	IF i16_anfangspos_mit_tzk[no] < 0 OR i16_endpos_mit_tzk[no] < 0 OR i16_anfangspos_mit_tzk[no] >= 360 OR i16_endpos_mit_tzk[no] >= 360 THEN
		 (* Fehlerfälle  mit Abbruch*)
		sm_positionseingabe := TRUE;
		EXIT; (* Schleifenabbruch *)
	ELSE (* Winkel sind o.k. und der Nocken wird bearbeitet -> ON/OFF *)
		sm_positionseingabe := FALSE;
		IF i16_anfangspos_mit_tzk[no] <> i16_endpos_mit_tzk[no] THEN
			(* Nocken setzen *)
			(* Anfangswinkel ist kleiner Endwinkel *)
			b_setzustand_anfang_kleiner_ende[no] := i16_anfangspos_mit_tzk[no] < i16_endpos_mit_tzk[no] AND
												i16_aktuelle_pos >= i16_anfangspos_mit_tzk[no] AND
												i16_aktuelle_pos <= i16_endpos_mit_tzk[no];
			(* Anfangswinkel ist grösser Endwinkel *)
			b_setzustand_anfang_groesser_ende[no] := i16_anfangspos_mit_tzk[no] > i16_endpos_mit_tzk[no] AND
												(i16_aktuelle_pos >= i16_anfangspos_mit_tzk[no] OR
												i16_aktuelle_pos <= i16_endpos_mit_tzk[no]);

			(* Nocken ist gültig, d.h. wurde von der Maschine oder Bediener aktiviert *)
			IF	arr_nocken[no].b_camvalid AND
				(b_setzustand_anfang_kleiner_ende[no] OR b_setzustand_anfang_groesser_ende[no]) AND
				((b_verfahrrichtung_positiv AND arr_nocken[no].b_eff_direction_pos) OR	(* positive Drehrichtung und positive Wirkrichtung ist freigegeben *)
				(b_verfahrrichtung_negativ AND arr_nocken[no].b_eff_direction_neg)) 		(* negative Drehrichtung und negative Wirkrichtung ist freigegeben *)
				THEN
					arr_nocken[no].b_nockenzustand := TRUE;
			END_IF

			(* Nocken zurücksetzen *)
			(* Anfangswinkel ist kleiner Endwinkel *)
			b_resetzustand_anfang_kleiner_ende[no] := i16_anfangspos_mit_tzk[no] < i16_endpos_mit_tzk[no] AND
													(i16_aktuelle_pos < i16_anfangspos_mit_tzk[no] OR
													i16_aktuelle_pos  > i16_endpos_mit_tzk[no]);
			(* Anfangswinkel ist grösser Endwinkel *)
			b_resetzustand_anfang_groesser_ende[no] := i16_anfangspos_mit_tzk[no] > i16_endpos_mit_tzk[no] AND
													i16_aktuelle_pos < i16_anfangspos_mit_tzk[no] AND
													i16_aktuelle_pos > i16_endpos_mit_tzk[no];

			(* Nocken ist ungültig, d.h. wurde von der Maschine oder Bediener deaktiviert *)
			IF	NOT arr_nocken[no].b_camvalid OR
				(b_resetzustand_anfang_kleiner_ende[no] OR b_resetzustand_anfang_groesser_ende[no])
				THEN
					arr_nocken[no].b_nockenzustand := FALSE;
			END_IF
		ELSE
			(* Anfang = Ende -> Nocken ist false *)
			arr_nocken[no].b_nockenzustand := FALSE;
		END_IF
	END_IF

	(* Aktive Nocken auf ihre Spuren setzen *)
	IF arr_nocken[no].b_camvalid AND arr_nocken[no].b_nockenzustand THEN
		arr_spur[arr_nocken[no].i16_track_no] := TRUE;
	END_IF
END_FOR

IF st_config.b_config_fertig THEN
	(* Fehlermeldungen und Betriebsmeldungen ab dem Startindex in die globalen Meldungsarrays schreiben *)
	garr_stoermeldungen[st_config.i16_meld_startindex + 0] := sm_positionseingabe;
	garr_stoermeldungen[st_config.i16_meld_startindex + 1] := sm_vorsteuerung;
	garr_stoermeldungen[st_config.i16_meld_startindex + 2] := FALSE;
	garr_stoermeldungen[st_config.i16_meld_startindex + 3] := FALSE;
	garr_stoermeldungen[st_config.i16_meld_startindex + 4] := FALSE;
	garr_stoermeldungen[st_config.i16_meld_startindex + 5] := FALSE;
	garr_stoermeldungen[st_config.i16_meld_startindex + 6] := FALSE;
	garr_stoermeldungen[st_config.i16_meld_startindex + 7] := FALSE;
	garr_stoermeldungen[st_config.i16_meld_startindex + 8] := FALSE;
	garr_stoermeldungen[st_config.i16_meld_startindex + 9] := FALSE;
	garr_stoermeldungen[st_config.i16_meld_startindex + 10] := FALSE;
	garr_stoermeldungen[st_config.i16_meld_startindex + 11] := FALSE;
	garr_stoermeldungen[st_config.i16_meld_startindex + 12] := FALSE;
	garr_stoermeldungen[st_config.i16_meld_startindex + 13] := FALSE;
	garr_stoermeldungen[st_config.i16_meld_startindex + 14] := FALSE;
	garr_stoermeldungen[st_config.i16_meld_startindex + 15] := FALSE;
	garr_stoermeldungen[st_config.i16_meld_startindex + 16] := FALSE;
	garr_stoermeldungen[st_config.i16_meld_startindex + 17] := FALSE;
	garr_stoermeldungen[st_config.i16_meld_startindex + 18] := FALSE;
	garr_stoermeldungen[st_config.i16_meld_startindex + 19] := FALSE;
	
	garr_betriebsmeldungen[st_config.i16_meld_startindex + 0] := FALSE;
	garr_betriebsmeldungen[st_config.i16_meld_startindex + 1] := FALSE;
	garr_betriebsmeldungen[st_config.i16_meld_startindex + 2] := FALSE;
	garr_betriebsmeldungen[st_config.i16_meld_startindex + 3] := FALSE;
	garr_betriebsmeldungen[st_config.i16_meld_startindex + 4] := FALSE;
	garr_betriebsmeldungen[st_config.i16_meld_startindex + 5] := FALSE;
	garr_betriebsmeldungen[st_config.i16_meld_startindex + 6] := FALSE;
	garr_betriebsmeldungen[st_config.i16_meld_startindex + 7] := FALSE;
	garr_betriebsmeldungen[st_config.i16_meld_startindex + 8] := FALSE;
	garr_betriebsmeldungen[st_config.i16_meld_startindex + 9] := FALSE;
	garr_betriebsmeldungen[st_config.i16_meld_startindex + 10] := FALSE;
	garr_betriebsmeldungen[st_config.i16_meld_startindex + 11] := FALSE;
	garr_betriebsmeldungen[st_config.i16_meld_startindex + 12] := FALSE;
	garr_betriebsmeldungen[st_config.i16_meld_startindex + 13] := FALSE;
	garr_betriebsmeldungen[st_config.i16_meld_startindex + 14] := FALSE;
	garr_betriebsmeldungen[st_config.i16_meld_startindex + 15] := FALSE;
	garr_betriebsmeldungen[st_config.i16_meld_startindex + 16] := FALSE;
	garr_betriebsmeldungen[st_config.i16_meld_startindex + 17] := FALSE;
	garr_betriebsmeldungen[st_config.i16_meld_startindex + 18] := FALSE;
	garr_betriebsmeldungen[st_config.i16_meld_startindex + 19] := FALSE;
END_IF
END_FUNCTION_BLOCK

(* POU EPT Lib/Funktionsbausteine/Nockenschaltwerke/NSW_LREAL/ST_Nockenschaltwerk_lreal, ST *)
FUNCTION_BLOCK ST_Nockenschaltwerk_lreal
VAR_INPUT
	r_achsposition							: LREAL;
	r_achsgeschwindigkeit						: LREAL;
	i16_verfahrrichtung_achse_extern			: INT;
	b_verfahrrichtungsauswertung_extern			: BOOL;
	i16_art_der_achse							: enum_ecd_typ;
	st_config									: struct_config;
END_VAR
VAR_IN_OUT
	st_visu									: struct_visu;
	arr_nocken								: ARRAY [0..MAX_NOCKENGERUEST] OF struct_nocken_lreal;
END_VAR
VAR_OUTPUT
END_VAR
VAR
	b_first_cycle 								: BOOL := TRUE;
	r_aktuelle_pos 							: T_FIX16;
	r_alte_pos	 							: T_FIX16;
	b_verfahrrichtung_positiv 					: BOOL := FALSE;
	b_verfahrrichtung_negativ					: BOOL := FALSE;
	r_zeit_fuer_1einheit						: LREAL := 0.0;
	r_anfangspos_mit_tzk 						: ARRAY [0..MAX_NOCKENGERUEST] OF LREAL := 0.0;
	r_endpos_mit_tzk 							: ARRAY [0..MAX_NOCKENGERUEST] OF LREAL := 0.0;
	r_vorsteuerpos_max						: LREAL := 0.0;
	i16_verfahrrichtung_achse_intern				: INT := 0;
	sm_positionseingabe						: BOOL := FALSE;
	sm_vorsteuerung							: BOOL := FALSE;
	sp, no									: UINT := 0;
	arr_spur									: ARRAY [0..MAX_NOCKENGERUEST] OF BOOL;
	b_setzustand_anfang_kleiner_ende			: ARRAY [0..MAX_NOCKENGERUEST] OF BOOL;
	b_setzustand_anfang_groesser_ende		: ARRAY [0..MAX_NOCKENGERUEST] OF BOOL;
	b_resetzustand_anfang_kleiner_ende		: ARRAY [0..MAX_NOCKENGERUEST] OF BOOL;
	b_resetzustand_anfang_groesser_ende		: ARRAY [0..MAX_NOCKENGERUEST] OF BOOL;
END_VAR
(* Funktionsbaustein Nockenschaltwerk *)
(* Funktion für lineare und rotatorische Achsen *)
CASE i16_art_der_achse  OF
1:	(* Linearachse *)
	IF b_first_cycle THEN
		b_first_cycle := FALSE;

		(* Setze Drehrichtung Positiv. Da wenn beide Drehrichtungen nicht gesetzt sind, keine Nocke aktiv wird *)
		r_vorsteuerpos_max := 100.0;
		b_verfahrrichtung_positiv := TRUE;
		b_verfahrrichtung_negativ := FALSE;
		r_alte_pos := r_aktuelle_pos;
	END_IF

	(* Aktuelle Position für weitere Komponenten zur Verfügung stellen *)
	r_aktuelle_pos := LREAL_TO_FIX16(r_achsposition,2);

	(* Verfahrrichtung überwachen *)
	IF FIX16_TO_LREAL(r_aktuelle_pos) > FIX16_TO_LREAL(r_alte_pos) THEN
		i16_verfahrrichtung_achse_intern := 1;
		r_alte_pos := r_aktuelle_pos;
	ELSIF FIX16_TO_LREAL(r_aktuelle_pos) < FIX16_TO_LREAL(r_alte_pos) THEN
		i16_verfahrrichtung_achse_intern := -1;
		r_alte_pos := r_aktuelle_pos;
	END_IF

	IF b_verfahrrichtungsauswertung_extern THEN
		IF i16_verfahrrichtung_achse_extern = 1 THEN
			b_verfahrrichtung_positiv := TRUE;
			b_verfahrrichtung_negativ := FALSE;
		ELSIF i16_verfahrrichtung_achse_extern = -1 THEN
			b_verfahrrichtung_positiv := FALSE;
			b_verfahrrichtung_negativ := TRUE;
		END_IF
	ELSE
		IF i16_verfahrrichtung_achse_intern = 1 THEN
			b_verfahrrichtung_positiv := TRUE;
			b_verfahrrichtung_negativ := FALSE;
		ELSIF i16_verfahrrichtung_achse_intern = -1 THEN
			b_verfahrrichtung_positiv := FALSE;
			b_verfahrrichtung_negativ := TRUE;
		END_IF
	END_IF

	IF r_achsgeschwindigkeit >= 1.0 THEN
		r_zeit_fuer_1einheit := 0.001 * r_achsgeschwindigkeit;		(* REAL-Zahl in ms *)
	ELSE
		r_zeit_fuer_1einheit := 0.0;
	END_IF

	(* Totzeitkompensation durch Vorsteuerung *)
	FOR no := 0  TO SIZEOF (arr_nocken)/SIZEOF(arr_nocken[0]) -1 DO
		(* Berechnung der Vorsteuerposition *)
		 arr_nocken[no].r_vorsteuerpos :=  (TIME_TO_LREAL(arr_nocken[no].t_vorsteuerzeit)) * r_zeit_fuer_1einheit;
		IF  arr_nocken[no].r_vorsteuerpos >= r_vorsteuerpos_max THEN
			 arr_nocken[no].r_vorsteuerpos := 0.0;
			sm_vorsteuerung := TRUE;
		ELSE
			sm_vorsteuerung := FALSE;
		END_IF

		(* Nockentoleranz mit Berücksichtigung der Vorsteuerzeit für Anfangswinkel*)
		r_anfangspos_mit_tzk[no] := arr_nocken[no].r_cam_begin - arr_nocken[no].r_vorsteuerpos;
		(* Nockentoleranz mit Berücksichtigung der Vorsteuerzeit für Endwinkel*)
		r_endpos_mit_tzk[no] := arr_nocken[no].r_cam_end - arr_nocken[no].r_vorsteuerpos;

		IF r_anfangspos_mit_tzk[no] <> r_endpos_mit_tzk[no] THEN
			(* Nocken setzen *)
			(* Anfangsposition ist kleiner Endposition *)
			b_setzustand_anfang_kleiner_ende[no] := r_anfangspos_mit_tzk[no] < r_endpos_mit_tzk[no] AND
													FIX16_TO_LREAL(r_aktuelle_pos) >= r_anfangspos_mit_tzk[no] AND
													FIX16_TO_LREAL(r_aktuelle_pos) <= r_endpos_mit_tzk[no];
			(* Anfangsposition ist grösser Endposition *)
			b_setzustand_anfang_groesser_ende[no] := r_anfangspos_mit_tzk[no] > r_endpos_mit_tzk[no] AND
													FIX16_TO_LREAL(r_aktuelle_pos) <= r_anfangspos_mit_tzk[no] AND
													FIX16_TO_LREAL(r_aktuelle_pos) >= r_endpos_mit_tzk[no];
	
			(* Nocken ist gültig, d.h. wurde von der Maschine oder Bediener aktiviert *)
			IF	arr_nocken[no].b_camvalid AND
				(b_setzustand_anfang_kleiner_ende[no] OR b_setzustand_anfang_groesser_ende[no]) AND
				((b_verfahrrichtung_positiv AND arr_nocken[no].b_eff_direction_pos) OR	(* positive Drehrichtung und positive Wirkrichtung ist freigegeben *)
				(b_verfahrrichtung_negativ AND arr_nocken[no].b_eff_direction_neg)) 		(* negative Drehrichtung und negative Wirkrichtung ist freigegeben *)
				THEN
					arr_nocken[no].b_nockenzustand := TRUE;
			END_IF
	
			(* Nocken zurücksetzen *)
			(* Anfangswinkel ist kleiner Endwinkel *)
			b_resetzustand_anfang_kleiner_ende[no] := r_anfangspos_mit_tzk[no] < r_endpos_mit_tzk[no] AND
													(FIX16_TO_LREAL(r_aktuelle_pos) < r_anfangspos_mit_tzk[no] OR
													FIX16_TO_LREAL(r_aktuelle_pos)  > r_endpos_mit_tzk[no]);
			(* Anfangswinkel ist grösser Endwinkel *)
			b_resetzustand_anfang_groesser_ende[no] := r_anfangspos_mit_tzk[no] > r_endpos_mit_tzk[no] AND
													(FIX16_TO_LREAL(r_aktuelle_pos) > r_anfangspos_mit_tzk[no] OR
													FIX16_TO_LREAL(r_aktuelle_pos) < r_endpos_mit_tzk[no]);
	
			(* Nocken ist ungültig, d.h. wurde von der Maschine oder Bediener deaktiviert *)
			IF	NOT arr_nocken[no].b_camvalid OR
				b_resetzustand_anfang_kleiner_ende[no] OR
				b_resetzustand_anfang_groesser_ende[no] OR
				(* Zusatzbedingung für Nockenzustand rücksetzen ist nur bei Linearachsen sinnvoll *)
				(b_verfahrrichtung_positiv AND NOT arr_nocken[no].b_eff_direction_pos AND arr_nocken[no].b_eff_direction_neg) OR	(* positive Drehrichtung und positive Wirkrichtung ist freigegeben *)
				(b_verfahrrichtung_negativ AND NOT arr_nocken[no].b_eff_direction_neg AND arr_nocken[no].b_eff_direction_pos)		(* negative Drehrichtung und negative Wirkrichtung ist freigegeben *)
				THEN
					arr_nocken[no].b_nockenzustand := FALSE;
			END_IF
		ELSE
			(* Anfang = Ende -> Nocken ist false *)
			arr_nocken[no].b_nockenzustand := FALSE;
		END_IF
	END_FOR

	(* Erst alle Spuren reset *)
	FOR sp := 0  TO SIZEOF (arr_spur)-1 DO
		arr_spur[sp] :=FALSE;
	END_FOR
	
	(* Dann aktive Nocken auf ihre Spuren setzen *)
	FOR no := 0  TO SIZEOF (arr_nocken)/SIZEOF(arr_nocken[0])-1 DO
		IF arr_nocken[no].b_camvalid AND arr_nocken[no].b_nockenzustand THEN
			arr_spur[arr_nocken[no].i16_track_no] := TRUE;
		END_IF
	END_FOR

2:	(* Rotatorische Achse *)
	IF b_first_cycle THEN
		b_first_cycle := FALSE;

		(* Setze Drehrichtung Positiv. Da wenn beide Drehrichtungen nicht gesetzt sind, keine Nocke aktiv wird *)
		r_vorsteuerpos_max := 60.0;
		b_verfahrrichtung_positiv := TRUE;
		b_verfahrrichtung_negativ := FALSE;
		r_alte_pos := r_aktuelle_pos;
	END_IF

	(* Aktuelle Position für weitere Komponenten zur Verfügung stellen *)
	r_aktuelle_pos := LREAL_TO_FIX16(r_achsposition,2);

	(* Verfahrrichtung überwachen *)
	IF FIX16_TO_LREAL(r_aktuelle_pos) > FIX16_TO_LREAL(r_alte_pos) THEN
		i16_verfahrrichtung_achse_intern := 1;
		r_alte_pos := r_aktuelle_pos;
	ELSIF FIX16_TO_LREAL(r_aktuelle_pos) < FIX16_TO_LREAL(r_alte_pos) THEN
		i16_verfahrrichtung_achse_intern := -1;
		r_alte_pos := r_aktuelle_pos;
	END_IF

	IF b_verfahrrichtungsauswertung_extern THEN
		IF i16_verfahrrichtung_achse_extern = 1 THEN
			b_verfahrrichtung_positiv := TRUE;
			b_verfahrrichtung_negativ := FALSE;
		ELSIF i16_verfahrrichtung_achse_extern = -1 THEN
			b_verfahrrichtung_positiv := FALSE;
			b_verfahrrichtung_negativ := TRUE;
		END_IF
	ELSE
		IF i16_verfahrrichtung_achse_intern = 1 THEN
			b_verfahrrichtung_positiv := TRUE;
			b_verfahrrichtung_negativ := FALSE;
		ELSIF i16_verfahrrichtung_achse_intern = -1 THEN
			b_verfahrrichtung_positiv := FALSE;
			b_verfahrrichtung_negativ := TRUE;
		END_IF
	END_IF

	IF r_achsgeschwindigkeit >= 1.0 THEN
		(* 0.006 = 360Grad / (60sec * 1000ms) *)
		r_zeit_fuer_1einheit := 0.006 * r_achsgeschwindigkeit;	(* REAL-Zahl in ms *)
	ELSE
		r_zeit_fuer_1einheit := 0.0;
	END_IF

	(* Totzeitkompensation durch Vorsteuerung *)
	FOR no := 0  TO SIZEOF (arr_nocken)/SIZEOF(arr_nocken[0]) -1 DO
		(* Berechnung des Vorsteuerwinkels *)
		arr_nocken[no].r_vorsteuerpos :=  (TIME_TO_LREAL(arr_nocken[no].t_vorsteuerzeit)) * r_zeit_fuer_1einheit;
		IF  arr_nocken[no].r_vorsteuerpos >= r_vorsteuerpos_max THEN
			 arr_nocken[no].r_vorsteuerpos := 0.0;
			sm_vorsteuerung := TRUE;
		ELSE
			sm_vorsteuerung := FALSE;
		END_IF

		(* Nockentoleranz mit Berücksichtigung der Vorsteuerzeit für Anfangswinkel*)
		r_anfangspos_mit_tzk[no] := arr_nocken[no].r_cam_begin -  arr_nocken[no].r_vorsteuerpos;
		IF r_anfangspos_mit_tzk[no] > 360.0 THEN
			r_anfangspos_mit_tzk[no] := r_anfangspos_mit_tzk[no] - 360.0;
		ELSIF r_anfangspos_mit_tzk[no] < 0.0 THEN
			r_anfangspos_mit_tzk[no] := r_anfangspos_mit_tzk[no] + 360.0;
		END_IF
		(* Nockentoleranz mit Berücksichtigung der Vorsteuerzeit für Endwinkel*)
		r_endpos_mit_tzk[no] := arr_nocken[no].r_cam_end -  arr_nocken[no].r_vorsteuerpos;
		IF r_endpos_mit_tzk[no] > 360.0 THEN
			r_endpos_mit_tzk[no] := r_endpos_mit_tzk[no] - 360.0;
		ELSIF r_endpos_mit_tzk[no] < 0.0 THEN
			r_endpos_mit_tzk[no] := r_endpos_mit_tzk[no] + 360.0;
		END_IF
	
		IF r_anfangspos_mit_tzk[no] < 0.0 OR r_endpos_mit_tzk[no] < 0.0 OR r_anfangspos_mit_tzk[no] >= 360.0 OR r_endpos_mit_tzk[no] >= 360.0 THEN
			 (* Fehlerfälle  mit Abbruch*)
			sm_positionseingabe := TRUE;
			EXIT; (* Schleifenabbruch *)
		ELSE (* Winkel sind o.k. und der Nocken wird bearbeitet -> ON/OFF *)
			sm_positionseingabe := FALSE;
			IF r_anfangspos_mit_tzk[no] <> r_endpos_mit_tzk[no] THEN
				(* Nocken setzen *)
				(* Anfangswinkel ist kleiner Endwinkel *)
				b_setzustand_anfang_kleiner_ende[no] := r_anfangspos_mit_tzk[no] < r_endpos_mit_tzk[no] AND
													FIX16_TO_LREAL(r_aktuelle_pos) >= r_anfangspos_mit_tzk[no] AND
													FIX16_TO_LREAL(r_aktuelle_pos) <= r_endpos_mit_tzk[no];
				(* Anfangswinkel ist grösser Endwinkel *)
				b_setzustand_anfang_groesser_ende[no] := r_anfangspos_mit_tzk[no] > r_endpos_mit_tzk[no] AND
													(FIX16_TO_LREAL(r_aktuelle_pos) >= r_anfangspos_mit_tzk[no] OR
													FIX16_TO_LREAL(r_aktuelle_pos) <= r_endpos_mit_tzk[no]);

				(* Nocken ist gültig, d.h. wurde von der Maschine oder Bediener aktiviert *)
				IF	arr_nocken[no].b_camvalid AND
					(b_setzustand_anfang_kleiner_ende[no] OR b_setzustand_anfang_groesser_ende[no]) AND
					((b_verfahrrichtung_positiv AND arr_nocken[no].b_eff_direction_pos) OR	(* positive Drehrichtung und positive Wirkrichtung ist freigegeben *)
					(b_verfahrrichtung_negativ AND arr_nocken[no].b_eff_direction_neg)) 		(* negative Drehrichtung und negative Wirkrichtung ist freigegeben *)
					THEN
						arr_nocken[no].b_nockenzustand := TRUE;
				END_IF

				(* Nocken zurücksetzen *)
				(* Anfangswinkel ist kleiner Endwinkel *)
				b_resetzustand_anfang_kleiner_ende[no] := r_anfangspos_mit_tzk[no] < r_endpos_mit_tzk[no] AND
														(FIX16_TO_LREAL(r_aktuelle_pos) < r_anfangspos_mit_tzk[no] OR
														FIX16_TO_LREAL(r_aktuelle_pos)  > r_endpos_mit_tzk[no]);
				(* Anfangswinkel ist grösser Endwinkel *)
				b_resetzustand_anfang_groesser_ende[no] := r_anfangspos_mit_tzk[no] > r_endpos_mit_tzk[no] AND
														FIX16_TO_LREAL(r_aktuelle_pos) < r_anfangspos_mit_tzk[no] AND
														FIX16_TO_LREAL(r_aktuelle_pos) > r_endpos_mit_tzk[no];

				(* Nocken ist ungültig, d.h. wurde von der Maschine oder Bediener deaktiviert *)
				IF	NOT arr_nocken[no].b_camvalid OR
					(b_resetzustand_anfang_kleiner_ende[no] OR b_resetzustand_anfang_groesser_ende[no])
					THEN
						arr_nocken[no].b_nockenzustand := FALSE;
				END_IF
			ELSE
				(* Anfang = Ende -> Nocken ist false *)
				arr_nocken[no].b_nockenzustand := FALSE;
			END_IF
		END_IF
	END_FOR

	(* Erst alle Spuren reset *)
	FOR sp := 0  TO SIZEOF (arr_spur)-1 DO
		arr_spur[sp] :=FALSE;
	END_FOR

	(* Dann aktive Nocken auf ihre Spuren setzen *)
	FOR no := 0  TO SIZEOF (arr_nocken)/SIZEOF(arr_nocken[0])-1 DO
		IF arr_nocken[no].b_camvalid AND arr_nocken[no].b_nockenzustand THEN
			arr_spur[arr_nocken[no].i16_track_no] := TRUE;
		END_IF
	END_FOR
END_CASE

IF st_config.b_config_fertig THEN
	(* Fehlermeldungen und Betriebsmeldungen ab dem Startindex in die globalen Meldungsarrays schreiben *)
	garr_stoermeldungen[st_config.i16_meld_startindex + 0] := sm_positionseingabe;
	garr_stoermeldungen[st_config.i16_meld_startindex + 1] := sm_vorsteuerung;
	garr_stoermeldungen[st_config.i16_meld_startindex + 2] := FALSE;
	garr_stoermeldungen[st_config.i16_meld_startindex + 3] := FALSE;
	garr_stoermeldungen[st_config.i16_meld_startindex + 4] := FALSE;
	garr_stoermeldungen[st_config.i16_meld_startindex + 5] := FALSE;
	garr_stoermeldungen[st_config.i16_meld_startindex + 6] := FALSE;
	garr_stoermeldungen[st_config.i16_meld_startindex + 7] := FALSE;
	garr_stoermeldungen[st_config.i16_meld_startindex + 8] := FALSE;
	garr_stoermeldungen[st_config.i16_meld_startindex + 9] := FALSE;
	garr_stoermeldungen[st_config.i16_meld_startindex + 10] := FALSE;
	garr_stoermeldungen[st_config.i16_meld_startindex + 11] := FALSE;
	garr_stoermeldungen[st_config.i16_meld_startindex + 12] := FALSE;
	garr_stoermeldungen[st_config.i16_meld_startindex + 13] := FALSE;
	garr_stoermeldungen[st_config.i16_meld_startindex + 14] := FALSE;
	garr_stoermeldungen[st_config.i16_meld_startindex + 15] := FALSE;
	garr_stoermeldungen[st_config.i16_meld_startindex + 16] := FALSE;
	garr_stoermeldungen[st_config.i16_meld_startindex + 17] := FALSE;
	garr_stoermeldungen[st_config.i16_meld_startindex + 18] := FALSE;
	garr_stoermeldungen[st_config.i16_meld_startindex + 19] := FALSE;
	
	garr_betriebsmeldungen[st_config.i16_meld_startindex + 0] := FALSE;
	garr_betriebsmeldungen[st_config.i16_meld_startindex + 1] := FALSE;
	garr_betriebsmeldungen[st_config.i16_meld_startindex + 2] := FALSE;
	garr_betriebsmeldungen[st_config.i16_meld_startindex + 3] := FALSE;
	garr_betriebsmeldungen[st_config.i16_meld_startindex + 4] := FALSE;
	garr_betriebsmeldungen[st_config.i16_meld_startindex + 5] := FALSE;
	garr_betriebsmeldungen[st_config.i16_meld_startindex + 6] := FALSE;
	garr_betriebsmeldungen[st_config.i16_meld_startindex + 7] := FALSE;
	garr_betriebsmeldungen[st_config.i16_meld_startindex + 8] := FALSE;
	garr_betriebsmeldungen[st_config.i16_meld_startindex + 9] := FALSE;
	garr_betriebsmeldungen[st_config.i16_meld_startindex + 10] := FALSE;
	garr_betriebsmeldungen[st_config.i16_meld_startindex + 11] := FALSE;
	garr_betriebsmeldungen[st_config.i16_meld_startindex + 12] := FALSE;
	garr_betriebsmeldungen[st_config.i16_meld_startindex + 13] := FALSE;
	garr_betriebsmeldungen[st_config.i16_meld_startindex + 14] := FALSE;
	garr_betriebsmeldungen[st_config.i16_meld_startindex + 15] := FALSE;
	garr_betriebsmeldungen[st_config.i16_meld_startindex + 16] := FALSE;
	garr_betriebsmeldungen[st_config.i16_meld_startindex + 17] := FALSE;
	garr_betriebsmeldungen[st_config.i16_meld_startindex + 18] := FALSE;
	garr_betriebsmeldungen[st_config.i16_meld_startindex + 19] := FALSE;
END_IF
END_FUNCTION_BLOCK

(* POU EPT Lib/Funktionsbausteine/Nockenschaltwerke/NZW/ST_Nockenzaehlwerk, ST *)
FUNCTION_BLOCK ST_Nockenzaehlwerk
VAR_INPUT
	i16_wkz_vorbesetzwert		: INT;
	b_zustand_spur			: BOOL;
	b_externer_zaehler_reset	: BOOL;
END_VAR
VAR_OUTPUT
	b_aktionsnocken			: BOOL;
END_VAR
VAR
	fb_ctu_hubzaehler			: CTU;
	fb_r_trig_zaehler			: R_TRIG;
	fb_r_trig_ot_nocken		: R_TRIG;
	b_interner_zaehler_reset	: BOOL := FALSE;
END_VAR
(* Zählwerk für Aktionen, die OT-Nocken abhängig sind
Anwendung: Nacheiner bestimmten Anzahl von Umdrehungen soll eine Aktion ausgelöst werden.
Der Ausgang ist für eine Umdrehung aktiv, bevor er wieder zurückgesetzt wird. *)
fb_ctu_hubzaehler(
	CU:=  b_zustand_spur,
	RESET:= b_interner_zaehler_reset OR b_externer_zaehler_reset,
	PV:= i16_wkz_vorbesetzwert,
	Q=> ,
	CV=> );

fb_r_trig_zaehler(CLK:= fb_ctu_hubzaehler.Q, Q=> );

(* Abfrage des Zählerstatus und daraus resultierende Aktionen *)
IF fb_r_trig_zaehler.Q THEN (* Bei Zählerstand erreicht, Ausgang für eine Umdrehung setzen *)
	b_aktionsnocken := TRUE;
END_IF
IF NOT fb_ctu_hubzaehler.Q AND fb_r_trig_ot_nocken.Q THEN
	b_aktionsnocken := FALSE; (* Nach einer Umdrehung wird der Ausgang wieder rückgesetzt *)
END_IF

fb_r_trig_ot_nocken(CLK:= b_zustand_spur, Q=> );

IF NOT  b_zustand_spur AND fb_ctu_hubzaehler.Q THEN
	b_interner_zaehler_reset := TRUE; (* Wenn Zählerstand erreicht, dann Zähler nullen *)
ELSIF b_interner_zaehler_reset AND fb_ctu_hubzaehler.CV = 0 THEN
	b_interner_zaehler_reset := FALSE; (* Wenn Zähler genullt, dann wieder freigeben für erneutes Zählen *)
END_IF
END_FUNCTION_BLOCK

(* POU EPT Lib/Funktionsbausteine/ST_AnalogIn, ST *)
FUNCTION_BLOCK ST_AnalogIn
VAR_INPUT
	t_verzoegerung				: TIME;
	st_config						: struct_config;
END_VAR
VAR_OUTPUT
END_VAR
VAR
	b_error						: BOOL := FALSE;
	e_i16_sensor_delayed_value	: INT := 0;
	i16_anzeigewert_max			: INT := 16#7FFF;
	i16_anzeigewert_min			: INT := 16#0000;
	r_offset_skalierung			: INT := 16#0000;
	r_gain_skalierung				: INT := 16#0000;
	fb_abfragetakt				: ST_Blinker;
	fb_r_trig_abfragetakt			: R_TRIG;
	sm_overrange				: BOOL := FALSE;
	sm_underrange				: BOOL := FALSE;
	sm_limit1						: BOOL := FALSE;
	sm_limit2						: BOOL := FALSE;
	sm_error						: BOOL := FALSE;
	st_sensor					AT %I* :struct_analog_in;
END_VAR
(* Aufbereitung und Skalierung eines analogen Sensorwertes *)
i16_anzeigewert_max := 16#7FFF;

(* Verzögerte Abfrage des Analogwertes *)
fb_abfragetakt(
	b_start:= TRUE,
	 t_taktzeit_on:= t_verzoegerung,
	 t_taktzeit_off:= t_verzoegerung,
	b_blinker_out=> );

fb_r_trig_abfragetakt(CLK:= fb_abfragetakt.b_blinker_out, Q=> );

IF fb_r_trig_abfragetakt.Q THEN
	e_i16_sensor_delayed_value := st_sensor.e_i16_value;
END_IF

(* Fehlermeldungen der Analogkarte *)
sm_overrange := st_sensor.e_b_status_overrange;
sm_underrange := st_sensor.e_b_status_underrange;
sm_limit1	:= BYTE_TO_BOOL (st_sensor.e_by_status_limit1);
sm_limit2	 := BYTE_TO_BOOL (st_sensor.e_by_status_limit2);
sm_error	:= st_sensor.e_b_status_error;

b_error := sm_overrange OR sm_underrange OR sm_limit1 OR sm_limit2 OR sm_error;

IF st_config.b_config_fertig THEN
	(* Fehlermeldungen und Betriebsmeldungen ab dem Startindex in die globalen Meldungsarrays schreiben *)
	garr_stoermeldungen[st_config.i16_meld_startindex + 0] := sm_overrange;
	garr_stoermeldungen[st_config.i16_meld_startindex + 1] := sm_underrange;
	garr_stoermeldungen[st_config.i16_meld_startindex + 2] := sm_limit1;
	garr_stoermeldungen[st_config.i16_meld_startindex + 3] := sm_limit2;
	garr_stoermeldungen[st_config.i16_meld_startindex + 4] := sm_error;
	garr_stoermeldungen[st_config.i16_meld_startindex + 5] := FALSE;
	garr_stoermeldungen[st_config.i16_meld_startindex + 6] := FALSE;
	garr_stoermeldungen[st_config.i16_meld_startindex + 7] := FALSE;
	garr_stoermeldungen[st_config.i16_meld_startindex + 8] := FALSE;
	garr_stoermeldungen[st_config.i16_meld_startindex + 9] := FALSE;
	garr_stoermeldungen[st_config.i16_meld_startindex + 10] := FALSE;
	garr_stoermeldungen[st_config.i16_meld_startindex + 11] := FALSE;
	garr_stoermeldungen[st_config.i16_meld_startindex + 12] := FALSE;
	garr_stoermeldungen[st_config.i16_meld_startindex + 13] := FALSE;
	garr_stoermeldungen[st_config.i16_meld_startindex + 14] := FALSE;
	garr_stoermeldungen[st_config.i16_meld_startindex + 15] := FALSE;
	garr_stoermeldungen[st_config.i16_meld_startindex + 16] := FALSE;
	garr_stoermeldungen[st_config.i16_meld_startindex + 17] := FALSE;
	garr_stoermeldungen[st_config.i16_meld_startindex + 18] := FALSE;
	garr_stoermeldungen[st_config.i16_meld_startindex + 19] := FALSE;
	
	garr_betriebsmeldungen[st_config.i16_meld_startindex + 0] := FALSE;
	garr_betriebsmeldungen[st_config.i16_meld_startindex + 1] := FALSE;
	garr_betriebsmeldungen[st_config.i16_meld_startindex + 2] := FALSE;
	garr_betriebsmeldungen[st_config.i16_meld_startindex + 3] := FALSE;
	garr_betriebsmeldungen[st_config.i16_meld_startindex + 4] := FALSE;
	garr_betriebsmeldungen[st_config.i16_meld_startindex + 5] := FALSE;
	garr_betriebsmeldungen[st_config.i16_meld_startindex + 6] := FALSE;
	garr_betriebsmeldungen[st_config.i16_meld_startindex + 7] := FALSE;
	garr_betriebsmeldungen[st_config.i16_meld_startindex + 8] := FALSE;
	garr_betriebsmeldungen[st_config.i16_meld_startindex + 9] := FALSE;
	garr_betriebsmeldungen[st_config.i16_meld_startindex + 10] := FALSE;
	garr_betriebsmeldungen[st_config.i16_meld_startindex + 11] := FALSE;
	garr_betriebsmeldungen[st_config.i16_meld_startindex + 12] := FALSE;
	garr_betriebsmeldungen[st_config.i16_meld_startindex + 13] := FALSE;
	garr_betriebsmeldungen[st_config.i16_meld_startindex + 14] := FALSE;
	garr_betriebsmeldungen[st_config.i16_meld_startindex + 15] := FALSE;
	garr_betriebsmeldungen[st_config.i16_meld_startindex + 16] := FALSE;
	garr_betriebsmeldungen[st_config.i16_meld_startindex + 17] := FALSE;
	garr_betriebsmeldungen[st_config.i16_meld_startindex + 18] := FALSE;
	garr_betriebsmeldungen[st_config.i16_meld_startindex + 19] := FALSE;
END_IF
END_FUNCTION_BLOCK

(* POU EPT Lib/Funktionsbausteine/ST_AnalogOut, ST *)
FUNCTION_BLOCK ST_AnalogOut
VAR_INPUT
	r_digital_in					: REAL;
	st_config						: struct_config;
END_VAR
VAR_OUTPUT
END_VAR
VAR
	b_error						: BOOL := FALSE;
	i16_ausgabewert_max			: INT := 16#7FFF;
	i16_ausgabewert_min			: INT := 16#0;
	i16_offset_skalierung			: INT := 16#0;
	i16_gain_skalierung			: INT := 16#CCC;
	i16_analogwert				: INT := 0;
	sm_error						: BOOL := FALSE;
	i16_analog_out				AT %Q* : INT;
END_VAR
(* ===Ausgabe eines analogen Sollwertes an einen Aktor=== *)
(* Die Kalibrierung der Geraden sollte hier nicht geändert werden!
Der Ausgabe wert ist vom Format INT, somit wurde kalibriert auf den maximalen Endwert von 7FFF mit der Steigung CCC.
Der Offset dient zum Verschieben der Geraden, wenn bei Eingangswert 0 kein Analogwert von 0 erreicht wird. *)

IF st_config.b_station_aktiv THEN
	(* Skalieren des Analogwertes und Ausgabe an die Karte: y = gain*wert + offset *)
	i16_analogwert := REAL_TO_INT(INT_TO_REAL(i16_gain_skalierung) * r_digital_in + INT_TO_REAL(i16_offset_skalierung));
	
	IF i16_analogwert < i16_ausgabewert_min THEN
		i16_analog_out := i16_ausgabewert_min;
		b_error := TRUE;
	ELSIF i16_analogwert > i16_ausgabewert_max THEN
		i16_analog_out := i16_ausgabewert_max;
		b_error := TRUE;
	ELSE
		i16_analog_out := i16_analogwert;
		b_error := FALSE;
	END_IF
ELSE
	i16_analog_out := 0;
	b_error := FALSE;
END_IF

(* Fehlermeldung Bereich *)
sm_error := b_error;

IF st_config.b_config_fertig THEN
	(* Fehlermeldungen und Betriebsmeldungen ab dem Startindex in die globalen Meldungsarrays schreiben *)
	garr_stoermeldungen[st_config.i16_meld_startindex + 0] := sm_error;
	garr_stoermeldungen[st_config.i16_meld_startindex + 1] := FALSE;
	garr_stoermeldungen[st_config.i16_meld_startindex + 2] := FALSE;
	garr_stoermeldungen[st_config.i16_meld_startindex + 3] := FALSE;
	garr_stoermeldungen[st_config.i16_meld_startindex + 4] := FALSE;
	garr_stoermeldungen[st_config.i16_meld_startindex + 5] := FALSE;
	garr_stoermeldungen[st_config.i16_meld_startindex + 6] := FALSE;
	garr_stoermeldungen[st_config.i16_meld_startindex + 7] := FALSE;
	garr_stoermeldungen[st_config.i16_meld_startindex + 8] := FALSE;
	garr_stoermeldungen[st_config.i16_meld_startindex + 9] := FALSE;
	garr_stoermeldungen[st_config.i16_meld_startindex + 10] := FALSE;
	garr_stoermeldungen[st_config.i16_meld_startindex + 11] := FALSE;
	garr_stoermeldungen[st_config.i16_meld_startindex + 12] := FALSE;
	garr_stoermeldungen[st_config.i16_meld_startindex + 13] := FALSE;
	garr_stoermeldungen[st_config.i16_meld_startindex + 14] := FALSE;
	garr_stoermeldungen[st_config.i16_meld_startindex + 15] := FALSE;
	garr_stoermeldungen[st_config.i16_meld_startindex + 16] := FALSE;
	garr_stoermeldungen[st_config.i16_meld_startindex + 17] := FALSE;
	garr_stoermeldungen[st_config.i16_meld_startindex + 18] := FALSE;
	garr_stoermeldungen[st_config.i16_meld_startindex + 19] := FALSE;
	
	garr_betriebsmeldungen[st_config.i16_meld_startindex + 0] := FALSE;
	garr_betriebsmeldungen[st_config.i16_meld_startindex + 1] := FALSE;
	garr_betriebsmeldungen[st_config.i16_meld_startindex + 2] := FALSE;
	garr_betriebsmeldungen[st_config.i16_meld_startindex + 3] := FALSE;
	garr_betriebsmeldungen[st_config.i16_meld_startindex + 4] := FALSE;
	garr_betriebsmeldungen[st_config.i16_meld_startindex + 5] := FALSE;
	garr_betriebsmeldungen[st_config.i16_meld_startindex + 6] := FALSE;
	garr_betriebsmeldungen[st_config.i16_meld_startindex + 7] := FALSE;
	garr_betriebsmeldungen[st_config.i16_meld_startindex + 8] := FALSE;
	garr_betriebsmeldungen[st_config.i16_meld_startindex + 9] := FALSE;
	garr_betriebsmeldungen[st_config.i16_meld_startindex + 10] := FALSE;
	garr_betriebsmeldungen[st_config.i16_meld_startindex + 11] := FALSE;
	garr_betriebsmeldungen[st_config.i16_meld_startindex + 12] := FALSE;
	garr_betriebsmeldungen[st_config.i16_meld_startindex + 13] := FALSE;
	garr_betriebsmeldungen[st_config.i16_meld_startindex + 14] := FALSE;
	garr_betriebsmeldungen[st_config.i16_meld_startindex + 15] := FALSE;
	garr_betriebsmeldungen[st_config.i16_meld_startindex + 16] := FALSE;
	garr_betriebsmeldungen[st_config.i16_meld_startindex + 17] := FALSE;
	garr_betriebsmeldungen[st_config.i16_meld_startindex + 18] := FALSE;
	garr_betriebsmeldungen[st_config.i16_meld_startindex + 19] := FALSE;
END_IF
END_FUNCTION_BLOCK

(* POU EPT Lib/Funktionsbausteine/ST_Check_Modulopos, ST *)
FUNCTION ST_Check_Modulopos : BOOL
VAR_INPUT
	akt_pos		: LREAL;
	ziel_pos		: LREAL;
END_VAR
VAR
	lr_rest		: LREAL;
	lr_pos		: LREAL;
END_VAR
(* Funktion zum Überprüfen des MC_MoveModulo-Befehls wegen seltsamen Fahrens bei der Anzahl der Modulo Umdrehungen *)

		(* !!!nicht getestet !!! *)

lr_rest := LTRUNC(ziel_pos / 360);

IF lr_rest < 1 THEN
	ST_Check_Modulopos := TRUE;
ELSE
	lr_pos := ziel_pos - (lr_rest * 360);
	
	IF lr_pos >= akt_pos THEN
		ST_Check_Modulopos := TRUE;
	ELSE
		ST_Check_Modulopos := FALSE;
	END_IF
END_IF
END_FUNCTION

(* POU EPT Lib/Funktionsbausteine/ST_Flasher, ST *)
FUNCTION_BLOCK ST_Flasher
VAR_INPUT
	b_start 			: BOOL;
	t_taktzeit_aus 		: TIME;
END_VAR
VAR_OUTPUT
	b_flasher_out 		: BOOL;
END_VAR
VAR
	ton_on			: TON;
	ton_off			: TON;
END_VAR
ton_on(IN:=b_start AND NOT ton_off.Q , PT:=  t_taktzeit_aus, Q=>b_flasher_out , ET=> );
ton_off(IN:= ton_on.Q  , PT:= t#250ms, Q=> , ET=> );
END_FUNCTION_BLOCK

(* POU EPT Lib/Programmbausteine/Routing/ADS-Kommunikation/ReadAdsStruct, ST *)
FUNCTION_BLOCK ReadAdsStruct
VAR_INPUT
	b_Execute				: BOOL;
	b_Reset					: BOOL;
	AmsNetId				: STRING;
	Port						: UINT;
	s_SymbolName			: STRING;
	dw_DestAdr				: DWORD;
END_VAR
VAR_OUTPUT
	b_Busy					: BOOL;
	b_Done					: BOOL;
	b_Error					: BOOL;
	b_ErrorID				: UDINT;
END_VAR
VAR
	s_SymbolNameOld		: STRING;
	str_SymInfo				: SYMINFOSTRUCT;

	fb_read_symbolinfo		: PLC_ReadSymInfoByName;
	fb_ads_read				: ADSREAD;

	Done					: BOOL;
	fb_ton_quitt				: TON;
	fb_state_entry				: ST_StateEntry;
END_VAR
fb_ton_quitt(IN:= , PT:= t#1s, Q=> , ET=> );

fb_state_entry(
	i16_next_step:= , 
	i16_pos:= 1,
	s_debugtext:= ,
	E=> ,
	X=> ,
	i16_step=> ,
	i16_last_step=> );

CASE fb_state_entry.i16_step OF
(*=======================================================*)
	0:
		IF b_Execute THEN
			fb_state_entry.i16_next_step := 10;
		END_IF

(*=======================================================*)
	10:	(* Get Symbolinfo if necessary *)
		b_Busy := TRUE;
		IF str_SymInfo.idxGroup <> 0 AND s_SymbolName = s_SymbolNameOld THEN
			fb_state_entry.i16_next_step := 100;
		ELSE
			fb_state_entry.i16_next_step := 20;
		END_IF

(*=======================================================*)
	20:	(* Read Symbolinfo *)
		fb_read_symbolinfo.START := TRUE;
		IF fb_read_symbolinfo.BUSY THEN
			fb_state_entry.i16_next_step := 30;
		END_IF

(*=======================================================*)
	30:	(* Done or Error *)
		IF NOT fb_read_symbolinfo.BUSY THEN
			IF NOT fb_read_symbolinfo.ERR THEN
				fb_read_symbolinfo.START := FALSE;
				s_SymbolNameOld := s_SymbolName;
				fb_state_entry.i16_next_step := 100;
			ELSE
				b_Error := TRUE;
				b_ErrorID := fb_read_symbolinfo.ERRID;
				fb_state_entry.i16_next_step := 1000;
			END_IF
		END_IF

(*=======================================================*)
	100:	(* Read Symbol-Data *)
			fb_ads_read.READ := TRUE;
			IF fb_ads_read.BUSY THEN
				fb_state_entry.i16_next_step := 110;
			END_IF

(*=======================================================*)
	110:	(* Read is Busy *)
		IF NOT fb_ads_read.BUSY THEN
			IF NOT fb_ads_read.ERR THEN
				fb_ads_read.READ := FALSE;
				b_Done := TRUE;
				b_Busy := FALSE;
				fb_state_entry.i16_next_step := 120;
			ELSE
				b_Error := TRUE;
				b_ErrorID := fb_ads_read.ERRID;
				fb_state_entry.i16_next_step := 1000;
			END_IF
		END_IF

(*=======================================================*)
	120:	(* Read erfolgreich abgeschlossen *)
		IF NOT b_Execute THEN
			b_Done := FALSE;
			b_Busy := FALSE;
			fb_state_entry.i16_next_step := 0;
		END_IF;

(*=======================================================*)
	1000:	(* Fehler *)
		fb_read_symbolinfo.START := FALSE;
		fb_ads_read.READ := FALSE;

		IF b_Reset THEN
			fb_state_entry.i16_next_step := 0;
			b_Done := FALSE;
			b_Busy := FALSE;
			b_Error := FALSE;
			b_ErrorID := 0;
		END_IF

END_CASE

fb_state_entry(
	i16_next_step:= , 
	i16_pos:= 2,
	s_debugtext:= ,
	E=> , 
	X=> ,
	i16_step=> ,
	i16_last_step=> );

fb_read_symbolinfo(
	NETID:= AmsNetId,
	PORT:= Port,
	SYMNAME:= s_SymbolName,
	START:= , 
	TMOUT:= DEFAULT_ADS_TIMEOUT,
	BUSY=> , 
	ERR=> , 
	ERRID=> , 
	SYMINFO=> str_SymInfo);

fb_ads_read(
	NETID:= AmsNetId,
	PORT:= Port,
	IDXGRP:= str_SymInfo.idxGroup,
	IDXOFFS:= str_SymInfo.idxOffset,
	LEN:= str_SymInfo.byteSize,
	DESTADDR:= dw_DestAdr,
	READ:= , 
	TMOUT:= DEFAULT_ADS_TIMEOUT,
	BUSY=> , 
	ERR=> , 
	ERRID=> );
END_FUNCTION_BLOCK

(* POU EPT Lib/Programmbausteine/Routing/ADS-Kommunikation/ST_ADS_Kommunikation, ST *)
FUNCTION_BLOCK ST_ADS_Kommunikation
VAR_INPUT
	s_read_symbol_name			: STRING;
	s_write_symbol_name			: STRING;
	dw_read_source_adr_vorher	: struct_station_vorher_out;
	dw_write_source_adr_vorher	: struct_station_vorher_in;
	dw_read_source_adr_nachher	: struct_station_nachher_out;
	dw_write_source_adr_nachher	: struct_station_nachher_in;
END_VAR
VAR
	fb_read_ads					: ReadAdsStruct;
	fb_write_ads					: WriteAdsStruct;

	fb_ton_wz					: TON;
	fb_ton_quitt					: TON;
	fb_state_entry					: ST_StateEntry;
	b_ibn_start					: BOOL := FALSE;
	fb_r_trig_ibn_start				: R_TRIG;
	fb_ton_ibn_start				: TON;
	s_AMSNetId					: STRING;
END_VAR
(* Zeiten *)
fb_ton_wz(IN:= , PT:= , Q=> , ET=> );
fb_ton_quitt(IN:= , PT:= t#3s, Q=> , ET=> );

fb_r_trig_ibn_start(CLK:= b_ibn_start, Q=> );
fb_ton_ibn_start(IN:= , PT:= t#1s, Q=> , ET=> );

IF fb_r_trig_ibn_start.Q THEN
	fb_ton_ibn_start.IN := TRUE;
ELSE
	IF fb_ton_ibn_start.Q THEN
		b_ibn_start := FALSE;
	 	fb_ton_ibn_start.IN := FALSE;
	END_IF
END_IF

fb_state_entry(
	i16_next_step:= , 
	i16_pos:= 1,
	s_debugtext:= ,
	E=> ,
	X=> ,
	i16_step=> ,
	i16_last_step=> );

CASE fb_state_entry.i16_step OF
(*=======================================================*)
	0:	(* Initialisierung *)
		fb_read_ads.b_Execute := FALSE;
		fb_write_ads.b_Execute := FALSE;
		fb_read_ads.b_Reset := FALSE;
		fb_write_ads.b_Reset := FALSE;
		fb_ton_wz.IN := FALSE;
		fb_state_entry.i16_next_step := 10;

(*=======================================================*)
	10:	(* Warte bis Routing-Verbindung zum Front-PC wurde angelegt wurde *)
		IF fb_state_entry.E THEN
			;
		END_IF

		(*-----------------------Weiterschaltbedingungen----------------------------*)
		IF ST_RoutingBackpanel.fb_state_entry.i16_step = 999 THEN
			fb_state_entry.i16_next_step := 20;
		END_IF

(*=======================================================*)
	20:	(* Lese NetId von angeschlossenen Remote-PCs *)
		IF fb_state_entry.E THEN
			s_AMSNetId :=  ST_RoutingBackpanel.s_backpanel_netid;
		END_IF

		fb_state_entry.i16_next_step := 100;

(*==========================LESEN=============================*)
	100:	(* Lesen der Symbole über ADS *)
		IF fb_state_entry.E THEN
			fb_read_ads.b_Execute := TRUE;
		END_IF

		IF fb_read_ads.b_Busy THEN
			fb_read_ads.b_Execute := FALSE;
			fb_state_entry.i16_next_step := 110;
		END_IF

(*=======================================================*)
	110:	(* Lesen abgeschlossen *)
		IF NOT fb_read_ads.b_Busy AND fb_read_ads.b_Done THEN
			fb_state_entry.i16_next_step := 200;
		ELSIF fb_read_ads.b_Error THEN
			fb_state_entry.i16_next_step := 1000;
		END_IF

(*===========================SCHREIBEN============================*)
	200:	(* Schreiben der Symbole über ADS *)
		IF fb_state_entry.E THEN
			fb_write_ads.b_Execute := TRUE;
		END_IF

		IF fb_write_ads.b_Busy THEN
			fb_write_ads.b_Execute := FALSE;
			fb_state_entry.i16_next_step := 210;
		END_IF

(*=======================================================*)
	210:	(* Schreiben abgeschlossen *)
		IF NOT fb_write_ads.b_Busy AND fb_write_ads.b_Done THEN
			fb_state_entry.i16_next_step := 999;
		ELSIF fb_write_ads.b_Error THEN
			fb_state_entry.i16_next_step := 1000;
		END_IF

(*=======================================================*)
	999:	(* Ende *)
		fb_state_entry.i16_next_step := 100;

(*=======================================================*)
	1000:	(* Fehler *)
		IF fb_state_entry.E THEN
			fb_read_ads.b_Execute := FALSE;
			fb_write_ads.b_Execute := FALSE;
			fb_ton_wz.IN := FALSE;
			fb_ton_quitt.IN := TRUE;
		END_IF

		IF  fb_ton_quitt.Q THEN
			fb_ton_quitt.IN := FALSE;
			fb_read_ads.b_Reset := TRUE;
			fb_write_ads.b_Reset := TRUE;
			fb_state_entry.i16_next_step := 0;
		END_IF
END_CASE

fb_state_entry(
	i16_next_step:= , 
	i16_pos:= 2,
	s_debugtext:= ,
	E=> , 
	X=> ,
	i16_step=> ,
	i16_last_step=> );

fb_read_ads(
	b_Execute:= ,
	b_Reset:= ,
	AmsNetId:= s_AMSNetId ,
	Port:= 801,
	s_SymbolName:=s_read_symbol_name ,
	dw_DestAdr:= ADR(dw_read_source_adr_vorher),
	b_Busy=> ,
	b_Done=> ,
	b_Error=> ,
	b_ErrorID=> );

fb_write_ads(
	b_Execute:= ,
	b_Reset:= ,
	AmsNetId:= s_AMSNetId,
	Port:= 801 ,
	s_SymbolName:=  s_write_symbol_name,
	dw_SourceAdr:= ADR(dw_write_source_adr_vorher) ,
	b_Busy=> ,
	b_Done=> ,
	b_Error=> ,
	b_ErrorID=> );
END_FUNCTION_BLOCK

(* POU EPT Lib/Programmbausteine/Routing/ADS-Kommunikation/WriteAdsStruct, ST *)
FUNCTION_BLOCK WriteAdsStruct
VAR_INPUT
	b_Execute				: BOOL;
	b_Reset					: BOOL;
	AmsNetId				: STRING;
	Port						: UINT;
	s_SymbolName			: STRING;
	dw_SourceAdr			: DWORD;
END_VAR
VAR_OUTPUT
	b_Busy					: BOOL;
	b_Done					: BOOL;
	b_Error					: BOOL;
	b_ErrorID				: UDINT;
END_VAR
VAR
	s_SymbolNameOld		: STRING;
	str_SymInfo				: SYMINFOSTRUCT;

	fb_read_symbolinfo		: PLC_ReadSymInfoByName;
	fb_ads_write				: ADSWRITE;

	Done					: BOOL;
	fb_ton_quitt				: TON;
	fb_state_entry				: ST_StateEntry;
END_VAR
fb_ton_quitt(IN:= , PT:= t#1s, Q=> , ET=> );

fb_state_entry(
	i16_next_step:= , 
	i16_pos:= 1,
	s_debugtext:= ,
	E=> ,
	X=> ,
	i16_step=> ,
	i16_last_step=> );

CASE fb_state_entry.i16_next_step OF
(*=======================================================*)
	0:
		IF b_Execute THEN
			fb_state_entry.i16_next_step := 10;
		END_IF

(*=======================================================*)
	10:	(* Get Symbolinfo if necessary *)
		b_Busy := TRUE;
		IF str_SymInfo.idxGroup <> 0 AND s_SymbolName = s_SymbolNameOld THEN
			fb_state_entry.i16_next_step := 100;
		ELSE
			fb_state_entry.i16_next_step := 20;
		END_IF

(*=======================================================*)
	20:	(* Read Symbolinfo *)
		fb_read_symbolinfo.START := TRUE;
		IF fb_read_symbolinfo.BUSY THEN
			fb_state_entry.i16_next_step := 30;
		END_IF

(*=======================================================*)
	30:	(* Done or Error *)
		IF NOT fb_read_symbolinfo.BUSY THEN
			IF NOT fb_read_symbolinfo.ERR THEN
				fb_read_symbolinfo.START := FALSE;
				s_SymbolNameOld := s_SymbolName;
				fb_state_entry.i16_next_step := 100;
			ELSE
				b_Error := TRUE;
				b_ErrorID := fb_read_symbolinfo.ERRID;
				fb_state_entry.i16_next_step := 1000;
			END_IF
		END_IF

(*=======================================================*)
	100:	(* Read Symbol-Data *)
			fb_ads_write.WRITE := TRUE;
			IF fb_ads_write.BUSY THEN
				fb_state_entry.i16_next_step := 110;
			END_IF

(*=======================================================*)
	110:	(* Read is Busy *)
		IF NOT fb_ads_write.BUSY THEN
			IF NOT fb_ads_write.ERR THEN
				fb_ads_write.WRITE := FALSE;
				b_Done := TRUE;
				b_Busy := FALSE;
				fb_state_entry.i16_next_step := 120;
			ELSE
				b_Error := TRUE;
				b_ErrorID := fb_ads_write.ERRID;
				fb_state_entry.i16_next_step := 1000;
			END_IF
		END_IF

(*=======================================================*)
	120:	(* Read erfolgreich abgeschlossen *)
		IF NOT b_Execute THEN
			b_Done := FALSE;
			b_Busy := FALSE;
			fb_state_entry.i16_next_step := 0;
		END_IF;

(*=======================================================*)
	1000:	(* Fehler *)
		fb_read_symbolinfo.START := FALSE;
		fb_ads_write.WRITE := FALSE;

		IF b_Reset THEN
			fb_state_entry.i16_next_step := 0;
			b_Done := FALSE;
			b_Busy := FALSE;
			b_Error := FALSE;
			b_ErrorID := 0;
		END_IF

END_CASE

fb_state_entry(
	i16_next_step:= , 
	i16_pos:= 2,
	s_debugtext:= ,
	E=> , 
	X=> ,
	i16_step=> ,
	i16_last_step=> );

fb_read_symbolinfo(
	NETID:= AmsNetId,
	PORT:= Port,
	SYMNAME:= s_SymbolName,
	START:= , 
	TMOUT:= DEFAULT_ADS_TIMEOUT,
	BUSY=> , 
	ERR=> , 
	ERRID=> , 
	SYMINFO=> str_SymInfo);

fb_ads_write(
	NETID:= AmsNetId,
	PORT:= Port,
	IDXGRP:= str_SymInfo.idxGroup,
	IDXOFFS:= str_SymInfo.idxOffset,
	LEN:= str_SymInfo.byteSize,
	SRCADDR:= dw_SourceAdr,
	WRITE:= ,
	TMOUT:= DEFAULT_ADS_TIMEOUT,
	BUSY=> , 
	ERR=> , 
	ERRID=> );
END_FUNCTION_BLOCK

(* POU EPT Lib/Programmbausteine/ST_Start_Batchscript, ST *)
FUNCTION_BLOCK ST_Start_Batchscript
VAR_INPUT
	bExecute			: BOOL;
	bQuit				: BOOL;
	st_pfad				: STRING;
END_VAR
VAR_OUTPUT
	bBusy				: BOOL;
	bReady				: BOOL;
	bError				: BOOL;
	nErrId				: UDINT;
END_VAR
VAR
	fb_ton_quitt					: TON;
	fb_state_entry					: ST_StateEntry;
	fb_r_trig_execute				: R_TRIG;
	fb_nt_start_process			: NT_StartProcess;
END_VAR
(* Starten eines Batchscriptes auf dem lokalen PC *)
fb_r_trig_execute(CLK:= bExecute, Q=> );
fb_ton_quitt(IN:= , PT:= t#100ms, Q=> , ET=> );

fb_state_entry(
	i16_next_step:= ,
	i16_pos:= 1,
	s_debugtext:= ,
	E=> ,
	X=> , 
	i16_step=> ,
	i16_last_step=> );

CASE fb_state_entry.i16_step OF
(*=======================================================*)
	0:(* INIT *)
		bBusy := FALSE;
		bReady := FALSE;
		bError := FALSE;
		nErrId := 0;
		fb_nt_start_process.START := FALSE;
		fb_state_entry.i16_next_step := 10;

(*=======================================================*)
	10:	(* Warte auf Execute-Befehl *)

		IF fb_r_trig_execute.Q THEN
			bReady := FALSE;
			bBusy := TRUE;
			fb_state_entry.i16_next_step := 20;
		END_IF

(*=======================================================*)
	20:	(* Starte mit Ausführen des Batchscriptes *)
		IF fb_state_entry.E THEN
			fb_nt_start_process.START := TRUE;
		END_IF

		IF fb_nt_start_process.BUSY THEN
			fb_nt_start_process.START := FALSE;
			fb_state_entry.i16_next_step := 30;
		END_IF

(*=======================================================*)
	30:	(* Script wurde erfolgreich ausgeführt *)
		IF NOT fb_nt_start_process.BUSY THEN
			IF NOT fb_nt_start_process.ERR THEN
				bBusy := FALSE;
				fb_state_entry.i16_next_step := 999;
			ELSE	(* Fehler *)
				fb_state_entry.i16_next_step := 1000;
			END_IF
		END_IF

(*=======================================================*)
	999:	(* Fertig *)
		bReady := TRUE;
		fb_state_entry.i16_next_step := 10;

(*=======================================================*)
	1000: (* Fehler *)
		IF fb_state_entry.E THEN
			bBusy := FALSE;
			bReady := FALSE;
			bError := TRUE;
			fb_ton_quitt.IN := FALSE;
		END_IF

		(*-----------------------Weiterschaltbedingungen----------------------------*)
		IF bQuit AND NOT fb_state_entry.E THEN
			bError := FALSE;
			fb_ton_quitt.IN := TRUE;
		END_IF

		IF fb_ton_quitt.Q THEN
			fb_ton_quitt.IN := FALSE;
			fb_state_entry.i16_next_step := 0;
		END_IF
END_CASE

fb_state_entry(
	i16_next_step:= , 
	i16_pos:= 2,
	s_debugtext:= ,
	E=> ,
	X=> ,
	i16_step=> ,
	i16_last_step=> );

fb_nt_start_process(
	NETID:= '',
	PATHSTR:= st_pfad,
	DIRNAME:= , 
	COMNDLINE:= ,
	START:= ,
	TMOUT:= DEFAULT_ADS_TIMEOUT,
	BUSY=> ,
	ERR=> , 
	ERRID=> nErrId);
END_FUNCTION_BLOCK

(* POU EPT Lib/Serielle Kommunikation/ST_BalluffTagReader, ST *)
FUNCTION_BLOCK ST_BalluffTagReader
VAR_INPUT
	st_config						: struct_config;
	i16_addresse					: INT := 0;
	i16_anzahl_byte				: INT := 0;
	s_schreib_daten				: ARRAY [0..100] OF BYTE;
	st_ctrl_in						: struct_ctrl_in;
END_VAR
VAR_OUTPUT
	s_lese_daten					: ARRAY [0..100] OF BYTE;
	s_transp_serial_number		: STRING;
	st_ctrl_out					: struct_ctrl_out;
END_VAR
VAR
	fb_ton_wz					: TON;
	fb_ton_uez					: TON;
	fb_ton_quitt					: TON;
	fb_r_trig_lesen				: R_TRIG;
	fb_r_trig_schreiben			: R_TRIG;
	t_wz							: TIME := t#0ms;
	fb_state_entry					: ST_StateEntry;
	fb_r_trig_ibn_lesen			: R_TRIG;
	fb_r_trig_ibn_schreiben			: R_TRIG;
	fb_ton_ibn_lesen				: TON;
	fb_ton_ibn_schreiben			: TON;
	b_ibn_lesen					: BOOL := FALSE;
	b_ibn_schreiben				: BOOL := FALSE;
	sm_fehler_rfid_reader			: BOOL := FALSE;
	sm_kein_tag_erkannt			: BOOL := FALSE;

	(* Puffer für RS232*)
	RxBuffer						:ComBuffer;
	TxBuffer						:ComBuffer;
	EL6ComInData AT %I* 			:EL6inData22B;
	EL6ComOutData AT %Q*  		:EL6outData22B;
	fb_serial_line					: SerialLineControl ;

	(* RFID *)
	fb_RFID_Reader				: FB_RFIDReader;
	st_access_data				: ST_RFID_AccessData;
	eErrCodeRcv					: E_RFID_ErrCodeRcv_Balluff;

	e_tag_im_aktionsfeld			AT %I* : BOOL;
END_VAR
(* Zeiten *)
fb_ton_wz(IN:= , PT:= , Q=>  , ET=> );
fb_ton_uez(IN:= , PT:= , Q=>  , ET=> );
fb_ton_quitt(IN:= , PT:= t#100ms, Q=> , ET=> );
fb_r_trig_lesen(CLK:= st_ctrl_in.b_start_lesen, Q=> );
fb_r_trig_schreiben(CLK:= st_ctrl_in.b_start_schreiben, Q=> );

(* Inbetriebnahme *)
fb_r_trig_ibn_lesen(CLK:= b_ibn_lesen, Q=> );
fb_r_trig_ibn_schreiben(CLK:= b_ibn_schreiben, Q=> );
fb_ton_ibn_lesen(IN:= , PT:= t#1s, Q=> , ET=> );
fb_ton_ibn_schreiben(IN:= , PT:= t#1s, Q=> , ET=> );

IF fb_r_trig_ibn_lesen.Q THEN
	fb_ton_ibn_lesen.IN := TRUE;
ELSE
	IF fb_ton_ibn_lesen.Q THEN
		b_ibn_lesen := FALSE;
	 	fb_ton_ibn_lesen.IN := FALSE;
	END_IF
END_IF

IF fb_r_trig_ibn_schreiben.Q THEN
	fb_ton_ibn_schreiben.IN := TRUE;
ELSE
	IF fb_ton_ibn_schreiben.Q THEN
		b_ibn_schreiben := FALSE;
	 	fb_ton_ibn_schreiben.IN := FALSE;
	END_IF
END_IF


(* Toplevel *)(*
IF fb_state_entry.i16_next_step > INIT AND fb_state_entry.i16_next_step < FEHLER THEN
	IF fb_state_entry.i16_next_step < STOP THEN
		IF st_ctrl_in.b_stop THEN
			fb_state_entry.i16_next_step := STOP;
		END_IF
	END_IF
END_IF*)

(* ==================================Schrittkette================================ *)
fb_state_entry(
	i16_next_step:= ,
	i16_pos:= 1,
	s_debugtext:= ,
	E=> ,
	X=> , 
	i16_step=> ,
	i16_last_step=> );

CASE fb_state_entry.i16_step OF
(*=======================================================*)
	INIT_OBJ:
		fb_state_entry.i16_next_step := INIT;

(*=======================================================*)
	INIT:
		IF fb_state_entry.E THEN
			fb_ton_wz.IN := FALSE;
			fb_ton_uez.IN := FALSE;
			fb_ton_quitt.IN := FALSE;
			sm_fehler_rfid_reader := FALSE;
			sm_kein_tag_erkannt := FALSE;
			fb_RFID_Reader.bExecute := FALSE;
			st_ctrl_out.b_fehler := FALSE;
			st_ctrl_out.b_bereit := FALSE;
			st_ctrl_out.b_fertig := FALSE;
		END_IF

		(*-----------------------Weiterschaltbedingungen----------------------------*)
(*		IF st_ctrl_in.b_init THEN*)
			fb_state_entry.i16_next_step := 20;
(*		END_IF*)

(*=======================================================*)
	20:	(* Reset Reader *)
		IF fb_state_entry.E THEN
			fb_RFID_Reader.bExecute := TRUE;
			fb_RFID_Reader.eCommand := eRFC_ResetReader;
		END_IF
	
		(*-----------------------Weiterschaltbedingungen----------------------------*)
		IF fb_RFID_Reader.bBusy THEN
			fb_state_entry.i16_next_step := 30;
		END_IF

(*=======================================================*)
	30:

		(*-----------------------Weiterschaltbedingungen----------------------------*)
		IF NOT fb_RFID_Reader.bBusy THEN
			fb_RFID_Reader.bExecute := FALSE;
			IF fb_RFID_Reader.bResponseRcv THEN
				fb_state_entry.i16_next_step := BEREIT;
			ELSIF  fb_RFID_Reader.bError THEN
				eErrCodeRcv := fb_RFID_Reader.iErrorID;
				sm_fehler_rfid_reader := TRUE;
				fb_state_entry.i16_next_step := FEHLER;
			END_IF
		END_IF

(*=======================================================*)
	BEREIT:
		IF fb_state_entry.E THEN
			st_ctrl_out.b_bereit := TRUE;
			st_ctrl_out.b_fertig := TRUE;
		END_IF

		IF fb_r_trig_lesen.Q OR fb_r_trig_ibn_lesen.Q THEN
			st_ctrl_out.b_fertig := FALSE;
			fb_state_entry.i16_next_step := 200;
		ELSIF fb_r_trig_schreiben.Q OR fb_r_trig_ibn_schreiben.Q THEN
			st_ctrl_out.b_fertig := FALSE;
			fb_state_entry.i16_next_step := 300;
		END_IF

(*=======================================================*)
	200: (* Abfrage, ob sich ein Tag im Aktionsfeld befindet, damit gelesen werden kann. *)
		IF fb_state_entry.E THEN
			fb_ton_uez.PT := t#1s;
			fb_ton_uez.IN := TRUE;
		END_IF

		(*-----------------------Weiterschaltbedingungen----------------------------*)
		IF e_tag_im_aktionsfeld THEN
			fb_ton_uez.IN := FALSE;
			fb_state_entry.i16_next_step := 210;
		ELSIF fb_ton_uez.Q THEN
			sm_kein_tag_erkannt := TRUE;
			fb_state_entry.i16_next_step := FEHLER;
		END_IF

(*=======================================================*)
	210: (* Start Lesen *)
		(* Vorbereiten Lesen *)
		IF fb_state_entry.E THEN
			fb_RFID_Reader.bExecute := TRUE;
			fb_RFID_Reader.eCommand := eRFC_ReadBlock;

			(* Datasize = blockCount * BlockSize *)
			st_access_data.iDataSize := i16_anzahl_byte;
			st_access_data.iBlockCount := i16_anzahl_byte;
			st_access_data.iBlockSize := 1;
			st_access_data.iStartBlock := i16_addresse;

			MEMSET(ADR(s_lese_daten), 0 , SIZEOF(s_lese_daten) );
			st_access_data.pData := ADR(s_lese_daten);
		END_IF

		(*-----------------------Weiterschaltbedingungen----------------------------*)
		IF fb_RFID_Reader.bBusy THEN
			fb_state_entry.i16_next_step := 220;
		END_IF

(*=======================================================*)
	220:	(* Fertig Lesen *)

		(*-----------------------Weiterschaltbedingungen----------------------------*)
		IF NOT fb_RFID_Reader.bBusy THEN
			fb_RFID_Reader.bExecute := FALSE;
			IF fb_RFID_Reader.bResponseRcv THEN
				fb_state_entry.i16_next_step := BEREIT;
			ELSIF  fb_RFID_Reader.bError THEN
				eErrCodeRcv := fb_RFID_Reader.iErrorID;
				sm_fehler_rfid_reader := TRUE;
				fb_state_entry.i16_next_step := FEHLER;
			END_IF
		END_IF

(*=======================================================*)
	300: (* Abfrage, ob sich ein Tag im Aktionsfeld befindet, damit geschrieben werden kann. *)
		IF fb_state_entry.E THEN
			fb_ton_uez.PT := t#1s;
			fb_ton_uez.IN := TRUE;
		END_IF

		(*-----------------------Weiterschaltbedingungen----------------------------*)
		IF e_tag_im_aktionsfeld THEN
			fb_ton_uez.IN := FALSE;
			fb_state_entry.i16_next_step := 310;
		ELSIF fb_ton_uez.Q THEN
			sm_kein_tag_erkannt := TRUE;
			fb_state_entry.i16_next_step := FEHLER;
		END_IF

(*=======================================================*)
	310: (* Start Schreiben *)
		(* Vorbereiten Schreiben *)
		IF fb_state_entry.E THEN
			fb_RFID_Reader.bExecute := TRUE;
			fb_RFID_Reader.eCommand := eRFC_WriteBlock;

			(* Datasize = blockCount * BlockSize *)
			st_access_data.iDataSize := i16_anzahl_byte;
			st_access_data.iBlockCount := i16_anzahl_byte;
			st_access_data.iBlockSize := 1;
			st_access_data.iStartBlock := i16_addresse;

			st_access_data.pData := ADR(s_schreib_daten);
		END_IF

		(*-----------------------Weiterschaltbedingungen----------------------------*)
		IF fb_RFID_Reader.bBusy THEN
			fb_state_entry.i16_next_step := 320;
		END_IF

(*=======================================================*)
	320:	(* Fertig Schreiben *)

		(*-----------------------Weiterschaltbedingungen----------------------------*)
		IF NOT fb_RFID_Reader.bBusy THEN
			fb_RFID_Reader.bExecute := FALSE;
			IF fb_RFID_Reader.bResponseRcv THEN
				fb_state_entry.i16_next_step := BEREIT;
			ELSIF  fb_RFID_Reader.bError THEN
				eErrCodeRcv := fb_RFID_Reader.iErrorID;
				sm_fehler_rfid_reader := TRUE;
				fb_state_entry.i16_next_step := FEHLER;
			END_IF
		END_IF

(*=======================================================*)
	FEHLER:
		IF fb_state_entry.E THEN
			fb_RFID_Reader.bExecute := FALSE;
			st_ctrl_out.b_fehler := TRUE;
			fb_ton_quitt.IN := FALSE;
		END_IF

		(*-----------------------Weiterschaltbedingungen----------------------------*)
		IF st_ctrl_in.b_quitt AND NOT fb_state_entry.E THEN
			st_ctrl_out.b_fehler := FALSE;
			fb_ton_quitt.IN := TRUE;
		END_IF

		IF fb_ton_quitt.Q THEN
			fb_ton_quitt.IN := FALSE;
			fb_state_entry.i16_next_step := INIT;
		END_IF

(*=======================================================*)
	STOP:
		IF fb_state_entry.E THEN
			fb_ton_quitt.IN := FALSE;
		END_IF

		(*-----------------------Weiterschaltbedingungen----------------------------*)
		IF st_ctrl_in.b_quitt AND NOT fb_state_entry.E THEN
			fb_ton_quitt.IN := TRUE;
		END_IF

		IF fb_ton_quitt.Q THEN
			fb_ton_quitt.IN := FALSE;
			fb_state_entry.i16_next_step := INIT;
		END_IF
END_CASE

fb_state_entry(
	i16_next_step:= , 
	i16_pos:= 2,
	s_debugtext:= ,
	E=> , 
	X=> , 
	i16_step=> ,
	i16_last_step=> );

(* RFID FBs *)
fb_serial_line(
	Mode		:= SERIALLINEMODE_EL6_22B,
	pComIn		:= ADR(EL6ComInData),
	pComOut	:= ADR(EL6ComOutData),
	SizeComIn	:= SIZEOF(EL6ComInData),
	TxBuffer		:= TxBuffer,
	RxBuffer		:= RxBuffer
);

fb_RFID_Reader(
	bExecute:= , 
	eCommand:= ,
	stAccessData:= st_access_data ,
	stCtrl:= , 
	stCfg:= , 
	eManufacturer:= eRFRM_Balluff,
	tTimeOut:= , 
	RxBuffer:= RxBuffer,
	TxBuffer:= TxBuffer,
	bBusy=> , 
	bResponseRcv=> ,
	eResponse=> , 
	bError=> ,
	iErrorID=> , 
	iErrCodeRcv=> ,
	stReaderCfg=> , 
	stReaderInfo=> , 
	stTranspInfo=> , 
	stRawData=> );

s_transp_serial_number := fb_RFID_Reader.stTranspInfo.sSerialNumber;

IF st_config.b_config_fertig THEN
	(* Fehlermeldungen ab dem Startindex in das globale Störmeldungsarray schreiben *)
	garr_stoermeldungen[st_config.i16_meld_startindex + 0] := sm_fehler_rfid_reader;
	garr_stoermeldungen[st_config.i16_meld_startindex + 1] := sm_kein_tag_erkannt;
	garr_stoermeldungen[st_config.i16_meld_startindex + 2] := FALSE;
	garr_stoermeldungen[st_config.i16_meld_startindex + 3] := FALSE;
	garr_stoermeldungen[st_config.i16_meld_startindex + 4] := FALSE;
	garr_stoermeldungen[st_config.i16_meld_startindex + 5] := FALSE;
	garr_stoermeldungen[st_config.i16_meld_startindex + 6] := FALSE;
	garr_stoermeldungen[st_config.i16_meld_startindex + 7] := FALSE;
	garr_stoermeldungen[st_config.i16_meld_startindex + 8] := FALSE;
	garr_stoermeldungen[st_config.i16_meld_startindex + 9] := FALSE;
	garr_stoermeldungen[st_config.i16_meld_startindex + 10] := FALSE;
	garr_stoermeldungen[st_config.i16_meld_startindex + 11] := FALSE;
	garr_stoermeldungen[st_config.i16_meld_startindex + 12] := FALSE;
	garr_stoermeldungen[st_config.i16_meld_startindex + 13] := FALSE;
	garr_stoermeldungen[st_config.i16_meld_startindex + 14] := FALSE;
	garr_stoermeldungen[st_config.i16_meld_startindex + 15] := FALSE;
	garr_stoermeldungen[st_config.i16_meld_startindex + 16] := FALSE;
	garr_stoermeldungen[st_config.i16_meld_startindex + 17] := FALSE;
	garr_stoermeldungen[st_config.i16_meld_startindex + 18] := FALSE;
	garr_stoermeldungen[st_config.i16_meld_startindex + 19] := FALSE;
	
	(* Betriebsmeldungen *)
	garr_betriebsmeldungen[st_config.i16_meld_startindex + 0] := FALSE;
	garr_betriebsmeldungen[st_config.i16_meld_startindex + 1] := FALSE;
	garr_betriebsmeldungen[st_config.i16_meld_startindex + 2] := FALSE;
	garr_betriebsmeldungen[st_config.i16_meld_startindex + 3] := FALSE;
	garr_betriebsmeldungen[st_config.i16_meld_startindex + 4] := FALSE;
	garr_betriebsmeldungen[st_config.i16_meld_startindex + 5] := FALSE;
	garr_betriebsmeldungen[st_config.i16_meld_startindex + 6] := FALSE;
	garr_betriebsmeldungen[st_config.i16_meld_startindex + 7] := FALSE;
	garr_betriebsmeldungen[st_config.i16_meld_startindex + 8] := FALSE;
	garr_betriebsmeldungen[st_config.i16_meld_startindex + 9] := FALSE;
	garr_betriebsmeldungen[st_config.i16_meld_startindex + 10] := FALSE;
	garr_betriebsmeldungen[st_config.i16_meld_startindex + 11] := FALSE;
	garr_betriebsmeldungen[st_config.i16_meld_startindex + 12] := FALSE;
	garr_betriebsmeldungen[st_config.i16_meld_startindex + 13] := FALSE;
	garr_betriebsmeldungen[st_config.i16_meld_startindex + 14] := FALSE;
	garr_betriebsmeldungen[st_config.i16_meld_startindex + 15] := FALSE;
	garr_betriebsmeldungen[st_config.i16_meld_startindex + 16] := FALSE;
	garr_betriebsmeldungen[st_config.i16_meld_startindex + 17] := FALSE;
	garr_betriebsmeldungen[st_config.i16_meld_startindex + 18] := FALSE;
	garr_betriebsmeldungen[st_config.i16_meld_startindex + 19] := FALSE;
END_IF
END_FUNCTION_BLOCK

(* POU EPT Lib/Serielle Kommunikation/ST_BarcodeReader, ST *)
FUNCTION_BLOCK ST_BarcodeReader
VAR_INPUT
	st_config						: struct_config;
	st_ctrl_in						: struct_ctrl_in;
END_VAR
VAR_OUTPUT
	st_ctrl_out					: struct_ctrl_out;
	s_last_barcode				: STRING;
END_VAR
VAR
	fb_ton_wz					: TON;
	fb_ton_uez					: TON;
	fb_ton_quitt					: TON;
	t_wz							: TIME := t#0ms;
	fb_state_entry					: ST_StateEntry;

	(* RS232-Schnittstelle *)
	(* Hinweis: Datenpuffer vom Typ ComBuffer werden vom Anwender niemals direkt beschrieben oder gelesen,
	sondern dienen nur als Zwischenspeicher für die Kommunikationsbausteine. *)
	RxBuffer						: ComBuffer;
	TxBuffer						: ComBuffer;
	COM_in_data AT %I* 			: PcComInData; (*EL6inData22B;*)
	COM_out_data AT %Q*  		: PcComOutData; (*EL6outData22B;*)
	fb_com_port_control			: SerialLineControl;
	com_port_control_error			: BOOL := FALSE;
	com_port_control_error_id		: ComError_t;

	(* ReceiveString empfängt eine Zeichenkette von der mit der Eingangsvariablen RxBuffer korrespondierenden Schnittstelle
	und speichert sie in der Ausgangsvariablen ReceivedString. *)
	fb_receive					: ReceiveString;
	s_tmp_string					: STRING := '';
	s_barcode					: STRING := '';
	i16_receive_string_len			: INT := 0;
	i16_suffix_len					: INT := 0;
	receive_error_id				: ComError_t;
	b_receive_timeout				: BOOL := FALSE;
	t_receive_timeout				: TIME := t#0s;

	fb_trig_new_string				: R_TRIG;

	sm_fehler_seriel				: BOOL := FALSE;
	sm_fehler_string				: BOOL := FALSE;
END_VAR
(* Zeiten *)
fb_ton_wz(IN:= , PT:= , Q=>  , ET=> );
fb_ton_uez(IN:= , PT:= t#1000ms, Q=>  , ET=> );
fb_ton_quitt(IN:= , PT:= t#50ms, Q=> , ET=> );

(* Toplevel *)
IF fb_state_entry.i16_next_step > INIT AND fb_state_entry.i16_next_step < FEHLER THEN
(*
	IF fb_state_entry.i16_next_step < STOP THEN
		IF st_ctrl_in.b_stop THEN
			fb_state_entry.i16_next_step := STOP;
		END_IF
	END_IF
*)
	IF com_port_control_error OR receive_error_id > 0 THEN
		sm_fehler_seriel := TRUE;
		fb_state_entry.i16_next_step := FEHLER;
	END_IF
END_IF

(* ==================================Schrittkette================================ *)
fb_state_entry(
	i16_next_step:= , 
	i16_pos:= 1,
	s_debugtext:= ,
	E=> ,
	X=> ,
	i16_step=> ,
	i16_last_step=> );

CASE fb_state_entry.i16_step OF
(*=======================================================*)
	INIT_OBJ:
		fb_state_entry.i16_next_step := INIT;

(*=======================================================*)
	INIT:
		IF fb_state_entry.E THEN
			fb_ton_wz.IN := FALSE;
			fb_ton_uez.IN := FALSE;
			fb_ton_quitt.IN := FALSE;
			sm_fehler_seriel := FALSE;
			sm_fehler_string := FALSE;
			st_ctrl_out.b_fehler := FALSE;
			st_ctrl_out.b_bereit := FALSE;
			st_ctrl_out.b_fertig := FALSE;

			t_receive_timeout := t#1s;
			i16_suffix_len := 2;
		END_IF

		(*-----------------------Weiterschaltbedingungen----------------------------*)
		IF st_ctrl_in.b_init THEN
			fb_state_entry.i16_next_step := 20;
		END_IF

(*=======================================================*)
	20:	(* Reset Schnittstelle *)
		IF fb_state_entry.E THEN
			fb_receive.Reset := TRUE;
			fb_ton_wz.PT := t#100ms;
			fb_ton_wz.IN := TRUE;
		END_IF
	
		(*-----------------------Weiterschaltbedingungen----------------------------*)
		IF fb_ton_wz.Q THEN
			fb_receive.Reset := FALSE;
			fb_ton_wz.IN := FALSE;
			fb_state_entry.i16_next_step := BEREIT;
		END_IF

(*=======================================================*)
	BEREIT:	(* Warte auf neuen Barcode *)
		IF fb_state_entry.E THEN
			st_ctrl_out.b_bereit := TRUE;
			st_ctrl_out.b_fertig := TRUE;
		END_IF

		(*-----------------------Weiterschaltbedingungen----------------------------*)
		IF fb_receive.Busy THEN
			st_ctrl_out.b_fertig := FALSE;
			fb_state_entry.i16_next_step := 110;
		END_IF

(*=======================================================*)
	110: (* Barcode wurde eingelesen *)
		IF NOT fb_receive.Busy  THEN
			IF fb_receive.Error = COMERROR_NOERROR THEN
				s_last_barcode := s_barcode;
				fb_state_entry.i16_next_step := BEREIT;
			ELSE	(* Fehler *)
				sm_fehler_seriel := TRUE;
				fb_state_entry.i16_next_step := FEHLER;
			END_IF
		END_IF

(*=======================================================*)
	FEHLER:
		IF fb_state_entry.E THEN
			st_ctrl_out.b_fehler := TRUE;
			fb_ton_quitt.IN := FALSE;
		END_IF

		(*-----------------------Weiterschaltbedingungen----------------------------*)
		IF st_ctrl_in.b_quitt AND NOT fb_state_entry.E THEN
			st_ctrl_out.b_fehler := FALSE;
			fb_ton_quitt.IN := TRUE;
		END_IF

		IF fb_ton_quitt.Q THEN
			fb_ton_quitt.IN := FALSE;
			fb_state_entry.i16_next_step := INIT;
		END_IF

(*=======================================================*)
	STOP:
		IF fb_state_entry.E THEN
			fb_ton_quitt.IN := FALSE;
		END_IF

		(*-----------------------Weiterschaltbedingungen----------------------------*)
		IF st_ctrl_in.b_quitt AND NOT fb_state_entry.E THEN
			fb_ton_quitt.IN := TRUE;
		END_IF

		IF fb_ton_quitt.Q THEN
			fb_ton_quitt.IN := FALSE;
			fb_state_entry.i16_next_step := INIT;
		END_IF
END_CASE

fb_state_entry(
	i16_next_step:= , 
	i16_pos:= 2,
	s_debugtext:= ,
	E=> , 
	X=> ,
	i16_step=> ,
	i16_last_step=> );

(* Aufruf Baustein für serielle Kommunikation *)
fb_com_port_control(
	Mode:= SERIALLINEMODE_PC_COM_PORT,
	pComIn:= ADR(COM_in_data),			(* I/O data; see global variables *)
	pComOut:= ADR(COM_out_data),		(* I/O data; see global variables *)
	SizeComIn:= SIZEOF(COM_in_data),		(* I/O data; see global variables *)
	TxBuffer:= TxBuffer,					(* transmit buffer; see global variables *)
	RxBuffer:= RxBuffer,					(* receive buffer; see global variables *)
	Error=> com_port_control_error,
	ErrorID=> com_port_control_error_id);
(* =================================== *)

(* Routine für Strings empfangen *)
fb_receive(
	Prefix:= '',
	Suffix:= '$R$N',		(* RETURN*)
	Timeout:= t_receive_timeout,
	ReceivedString:= s_tmp_string,
	RXbuffer:= RxBuffer,
	StringReceived=> ,
	Busy=> ,
	Error=> receive_error_id,
	RxTimeout=> b_receive_timeout );

fb_trig_new_string(CLK  := fb_receive.StringReceived, Q=> );

IF fb_trig_new_string.Q THEN
	i16_receive_string_len:=LEN(s_tmp_string);
	s_barcode:=LEFT(s_tmp_string, i16_receive_string_len - i16_suffix_len); (* Delete Suffix *)
END_IF
(* ========================== *)

IF st_config.b_config_fertig THEN
	(* Fehlermeldungen ab dem Startindex in das globale Störmeldungsarray schreiben *)
	garr_stoermeldungen[st_config.i16_meld_startindex + 0] := sm_fehler_seriel;
	garr_stoermeldungen[st_config.i16_meld_startindex + 1] := sm_fehler_string;
	garr_stoermeldungen[st_config.i16_meld_startindex + 2] := FALSE;
	garr_stoermeldungen[st_config.i16_meld_startindex + 3] := FALSE;
	garr_stoermeldungen[st_config.i16_meld_startindex + 4] := FALSE;
	garr_stoermeldungen[st_config.i16_meld_startindex + 5] := FALSE;
	garr_stoermeldungen[st_config.i16_meld_startindex + 6] := FALSE;
	garr_stoermeldungen[st_config.i16_meld_startindex + 7] := FALSE;
	garr_stoermeldungen[st_config.i16_meld_startindex + 8] := FALSE;
	garr_stoermeldungen[st_config.i16_meld_startindex + 9] := FALSE;
	garr_stoermeldungen[st_config.i16_meld_startindex + 10] := FALSE;
	garr_stoermeldungen[st_config.i16_meld_startindex + 11] := FALSE;
	garr_stoermeldungen[st_config.i16_meld_startindex + 12] := FALSE;
	garr_stoermeldungen[st_config.i16_meld_startindex + 13] := FALSE;
	garr_stoermeldungen[st_config.i16_meld_startindex + 14] := FALSE;
	garr_stoermeldungen[st_config.i16_meld_startindex + 15] := FALSE;
	garr_stoermeldungen[st_config.i16_meld_startindex + 16] := FALSE;
	garr_stoermeldungen[st_config.i16_meld_startindex + 17] := FALSE;
	garr_stoermeldungen[st_config.i16_meld_startindex + 18] := FALSE;
	garr_stoermeldungen[st_config.i16_meld_startindex + 19] := FALSE;
	
	(* Betriebsmeldungen *)
	garr_betriebsmeldungen[st_config.i16_meld_startindex + 0] := FALSE;
	garr_betriebsmeldungen[st_config.i16_meld_startindex + 1] := FALSE;
	garr_betriebsmeldungen[st_config.i16_meld_startindex + 2] := FALSE;
	garr_betriebsmeldungen[st_config.i16_meld_startindex + 3] := FALSE;
	garr_betriebsmeldungen[st_config.i16_meld_startindex + 4] := FALSE;
	garr_betriebsmeldungen[st_config.i16_meld_startindex + 5] := FALSE;
	garr_betriebsmeldungen[st_config.i16_meld_startindex + 6] := FALSE;
	garr_betriebsmeldungen[st_config.i16_meld_startindex + 7] := FALSE;
	garr_betriebsmeldungen[st_config.i16_meld_startindex + 8] := FALSE;
	garr_betriebsmeldungen[st_config.i16_meld_startindex + 9] := FALSE;
	garr_betriebsmeldungen[st_config.i16_meld_startindex + 10] := FALSE;
	garr_betriebsmeldungen[st_config.i16_meld_startindex + 11] := FALSE;
	garr_betriebsmeldungen[st_config.i16_meld_startindex + 12] := FALSE;
	garr_betriebsmeldungen[st_config.i16_meld_startindex + 13] := FALSE;
	garr_betriebsmeldungen[st_config.i16_meld_startindex + 14] := FALSE;
	garr_betriebsmeldungen[st_config.i16_meld_startindex + 15] := FALSE;
	garr_betriebsmeldungen[st_config.i16_meld_startindex + 16] := FALSE;
	garr_betriebsmeldungen[st_config.i16_meld_startindex + 17] := FALSE;
	garr_betriebsmeldungen[st_config.i16_meld_startindex + 18] := FALSE;
	garr_betriebsmeldungen[st_config.i16_meld_startindex + 19] := FALSE;
END_IF
END_FUNCTION_BLOCK

(* POU EPT Lib/Zylinder/ST_Zylinder12V012346E, ST *)
FUNCTION_BLOCK ST_Zylinder12V012346E
VAR_INPUT
	st_config							: struct_zylinder_config;
	bw_nocken_zylinder_einfahren		: BOOL;
	bw_nocken_zylinder_ausfahren		: BOOL;
	uw_nocken_zylinder_einfahren		: BOOL;
	uw_nocken_zylinder_ausfahren		: BOOL;
	b_direkttaste_ausfahren			: BOOL;
	b_direkttaste_mittefahren			: BOOL;
	b_direkttaste_einfahren				: BOOL;
	st_ctrl_in							: struct_zylinder_ctrl_in;
	e_druckwaechter					: BOOL;
	i16_betriebsart					: enum_betriebsarten;
	b_no_gesteuert_im_norm_betrieb	: BOOL;
	b_masterachse_hand_dialog_aktiv	: BOOL;
END_VAR
VAR_IN_OUT
	st_visu							: struct_zylinder_visu;
END_VAR
VAR_OUTPUT
	st_ctrl_out						: struct_zylinder_ctrl_out;
	a_ventil_einfahren					AT %Q* : BOOL;
	a_ventil_ausfahren				AT %Q* : BOOL;
END_VAR
VAR
	b_first_cycle 						: BOOL := TRUE;
	i16_anzahl_sensoren				: INT := 0;
	i16_anzahl_spulen					: INT := 0;
	b_sensor_eingefahren_vorhanden	: BOOL := FALSE;
	b_sensor_ausgefahren_vorhanden	: BOOL := FALSE;
	b_mit_tzk							: BOOL := FALSE;
	b_nockengesteuert				: BOOL := FALSE;
	b_zustand_uw_nocken_einfahren	: BOOL := FALSE;
	b_zustand_uw_nocken_ausfahren	: BOOL := FALSE;
	st_tzk							: struct_totzeitkompensation;
	fb_ton_uz_fahren					: TON;
	fb_ton_uz_endlage1				: TON;
	fb_ton_uz_endlage2				: TON;
	fb_ton_uz_endlage3				: TON;
	fb_ton_uz_sensor1					: TON;
	fb_ton_uz_sensor2					: TON;
	fb_ton_uz_sensor3					: TON;
	fb_ton_einausfahren				: TON;
	fb_r_trig_ibn_ausfahren				: R_TRIG;
	fb_r_trig_ibn_einfahren				: R_TRIG;
	fb_r_trig_ibn_quit					: R_TRIG;
	fb_ton_ibn_ausfahren				: TON;
	fb_ton_ibn_einfahren				: TON;
	fb_ton_ibn_quit					: TON;
	fb_ton_quitt						: TON;
	st_sm							: struct_zylinder_meldungen;
	fb_state_entry						: ST_StateEntry;
	b_ibn_zylinder_ausfahren			: BOOL := FALSE;
	b_ibn_zylinder_einfahren			: BOOL := FALSE;
	b_ibn_zylinderfehler_quit			: BOOL := FALSE;

	e_sensor1_eingefahren			AT %I* : BOOL;
	e_sensor1_ausgefahren			AT %I* : BOOL;
	e_sensor2_eingefahren			AT %I* : BOOL;
	e_sensor2_ausgefahren			AT %I* : BOOL;
	e_sensor3_eingefahren			AT %I* : BOOL;
	e_sensor3_ausgefahren			AT %I* : BOOL;
	e_sensor_mittegefahren			AT %I* : BOOL;
	e_taste_einfahren					AT %I* : BOOL;
	e_taste_ausfahren					AT %I* : BOOL;
END_VAR
IF b_first_cycle THEN
	b_first_cycle := FALSE;
	st_ctrl_out.b_fehler := FALSE;
	st_ctrl_out.b_eingefahren := FALSE;
	st_ctrl_out.b_ausgefahren := FALSE;
	st_ctrl_out.b_gestoppt := FALSE;
	st_sm.b_zeit_ausfahren1:= FALSE;
	st_sm.b_zeit_einfahren1:= FALSE;
	st_sm.b_endlage1	:= FALSE;
	st_sm.b_sensor1:= FALSE;
	st_sm.b_zeit_ausfahren2 := FALSE;
	st_sm.b_zeit_einfahren2 := FALSE;
	st_sm.b_endlage2	:= FALSE;
	st_sm.b_sensor2 := FALSE;
	st_sm.b_zeit_ausfahren3 := FALSE;
	st_sm.b_zeit_einfahren3 := FALSE;
	st_sm.b_endlage3	:= FALSE;
	st_sm.b_sensor3 := FALSE;
	st_sm.b_winkel_ausfahren1:= FALSE;
	st_sm.b_winkel_einfahren1:= FALSE;
	st_sm.b_winkel_ausfahren2 := FALSE;
	st_sm.b_winkel_einfahren2 := FALSE;
	st_sm.b_winkel_ausfahren3 := FALSE;
	st_sm.b_winkel_einfahren3 := FALSE;
	st_sm.b_zyltyp_nicht_definiert := FALSE;
	st_sm.b_reserve1:= FALSE;
END_IF

(* Inbetriebnahme *)
fb_r_trig_ibn_ausfahren(CLK:= b_ibn_zylinder_ausfahren, Q=> );
fb_r_trig_ibn_einfahren(CLK:= b_ibn_zylinder_einfahren, Q=> );
fb_r_trig_ibn_quit(CLK:= b_ibn_zylinderfehler_quit, Q=> );
fb_ton_ibn_ausfahren(IN:= , PT:= t#1s, Q=> , ET=> );
fb_ton_ibn_einfahren(IN:= , PT:= t#1s, Q=> , ET=> );
fb_ton_ibn_quit(IN:= , PT:= t#1s, Q=> , ET=> );
fb_ton_quitt(IN:= , PT:= t#50ms, Q=> , ET=> );

IF fb_r_trig_ibn_ausfahren.Q THEN
	fb_ton_ibn_ausfahren.IN := TRUE;
ELSE
	IF fb_ton_ibn_ausfahren.Q THEN
		b_ibn_zylinder_ausfahren := FALSE;
	 	fb_ton_ibn_ausfahren.IN := FALSE;
	END_IF
END_IF

IF fb_r_trig_ibn_einfahren.Q THEN
	fb_ton_ibn_einfahren.IN := TRUE;
ELSE
	IF fb_ton_ibn_einfahren.Q THEN
		b_ibn_zylinder_einfahren := FALSE;
	 	fb_ton_ibn_einfahren.IN := FALSE;
	END_IF
END_IF

IF fb_r_trig_ibn_quit.Q THEN
	fb_ton_ibn_quit.IN := TRUE;
ELSE
	IF fb_ton_ibn_quit.Q THEN
		b_ibn_zylinderfehler_quit := FALSE;
	 	fb_ton_ibn_quit.IN := FALSE;
	END_IF
END_IF

(* Simulationssensoren für den Zylinderhandbetrieb *)
IF  	gi16_betriebsart = HAND AND
	st_visu.i16_nr_zyl_im_handbetrieb = st_config.i16_identnummer AND
	fb_state_entry.i16_step > INIT_OBJ
	THEN
		CASE i16_anzahl_sensoren OF
			0:
				st_visu.b_sensor_mittegefahren := e_sensor_mittegefahren;
				st_visu.enu_zustand := fb_state_entry.i16_step;
			1:
				st_visu.b_sensor_ausgefahren := e_sensor1_ausgefahren;
				st_visu.b_sensor_eingefahren := e_sensor1_eingefahren;
				st_visu.enu_zustand := fb_state_entry.i16_step;
			2:
				IF b_sensor_eingefahren_vorhanden AND b_sensor_ausgefahren_vorhanden THEN
					st_visu.b_sensor_ausgefahren := e_sensor1_ausgefahren;
					st_visu.b_sensor_eingefahren := e_sensor1_eingefahren;
					st_visu.b_sensor_mittegefahren := e_sensor_mittegefahren;
				ELSIF b_sensor_ausgefahren_vorhanden THEN
					st_visu.b_sensor_ausgefahren := e_sensor1_ausgefahren OR e_sensor2_ausgefahren;
				ELSIF b_sensor_eingefahren_vorhanden THEN
					st_visu.b_sensor_eingefahren := e_sensor1_eingefahren OR e_sensor2_eingefahren;
				END_IF
				st_visu.enu_zustand := fb_state_entry.i16_step;
			4:
				st_visu.b_sensor_ausgefahren := e_sensor1_ausgefahren AND e_sensor2_ausgefahren;
				st_visu.b_sensor_eingefahren := e_sensor1_eingefahren AND e_sensor2_eingefahren;
				st_visu.b_sensor_mittegefahren := e_sensor_mittegefahren;
				st_visu.enu_zustand := fb_state_entry.i16_step;
			6:
				st_visu.b_sensor_ausgefahren := e_sensor1_ausgefahren AND e_sensor2_ausgefahren AND e_sensor3_ausgefahren;
				st_visu.b_sensor_eingefahren := e_sensor1_eingefahren AND e_sensor2_eingefahren AND e_sensor3_eingefahren;
				st_visu.b_sensor_mittegefahren := e_sensor_mittegefahren;
				st_visu.enu_zustand := fb_state_entry.i16_step;
		END_CASE
END_IF

(* Überwachungszeiten *)
fb_ton_uz_fahren(IN:= , PT:= st_config.t_ueberwachungszeit, Q=>  , ET=> );
fb_ton_uz_endlage1(IN:= , PT:= t#100ms, Q=> , ET=> );
fb_ton_uz_endlage2(IN:= , PT:= t#100ms, Q=> , ET=> );
fb_ton_uz_endlage3(IN:= , PT:= t#100ms, Q=> , ET=> );
fb_ton_uz_sensor1(IN:= , PT:= t#100ms, Q=> , ET=> );
fb_ton_uz_sensor2(IN:= , PT:= t#100ms, Q=> , ET=> );
fb_ton_uz_sensor3(IN:= , PT:= t#100ms, Q=> , ET=> );

(* Aus- und Einfahrzeit *)
fb_ton_einausfahren(IN:= , PT:= st_config.t_ein_aus_fahrzeit, Q=> , ET=> );

(* Totzeitkompensationszeit *)
st_tzk.fb_ton_tzk(IN:= , PT:= st_tzk.t_kompensationszeit, Q=> , ET=> );

IF fb_state_entry.i16_step > ZYL_INIT AND fb_state_entry.i16_step < ZYL_FEHLER THEN
	IF 	st_ctrl_in.b_stop AND
		(st_visu.i16_nr_zyl_im_handbetrieb <> st_config.i16_identnummer OR gi16_betriebsart <> HAND)
		THEN
			fb_state_entry.i16_next_step := GESTOPPT;
	END_IF
END_IF

(* Zylinder bewegen über Direkttasten von der hinteren Bedienoberfläche und Hardwaretaster *)
IF (b_direkttaste_ausfahren AND NOT b_direkttaste_einfahren) OR (e_taste_ausfahren AND NOT e_taste_einfahren) THEN
	fb_state_entry.i16_next_step := DIREKT_AUSFAHREN;
ELSIF (b_direkttaste_einfahren AND NOT b_direkttaste_ausfahren) OR (NOT e_taste_ausfahren AND e_taste_einfahren) THEN
	fb_state_entry.i16_next_step := DIREKT_EINFAHREN;
END_IF

(* ==================================Schrittkette================================ *)
fb_state_entry(
	i16_next_step:= ,
	i16_pos:= 1,
	s_debugtext:= ,
	E=> ,
	X=> ,
	i16_step=> ,
	i16_last_step=> );

CASE fb_state_entry.i16_step OF
	INIT_OBJ:	(* Zylindertyp feststellen *)
		IF st_config.b_config_fertig THEN
			(* Anzahl Spulen *)
			i16_anzahl_spulen := STRING_TO_INT(MID(st_config.str_zylinder_typ, 1, 1));
			(* Anzahl Sensoren *)
			i16_anzahl_sensoren := STRING_TO_INT(MID(st_config.str_zylinder_typ, 1, 3));
			(* Zylinder ist nockengesteuert *)
			IF FIND(st_config.str_zylinder_typ, 'NO') = 0 THEN
				b_nockengesteuert := FALSE;
			ELSE
				b_nockengesteuert := TRUE;
			END_IF
			(* Zylinder ist mit Totzeitkompensation *)
			IF FIND(st_config.str_zylinder_typ, 'TZK') = 0 THEN
				b_mit_tzk := FALSE;
			ELSE
				b_mit_tzk := TRUE;
			END_IF
			(* Vorhandene Sensoren *)
			IF FIND(st_config.str_zylinder_typ, 'AUS') >= 5 THEN
				b_sensor_ausgefahren_vorhanden := TRUE;
			ELSE
				b_sensor_ausgefahren_vorhanden := FALSE;
			END_IF
			IF FIND(st_config.str_zylinder_typ, 'EIN') >= 5 THEN
				b_sensor_eingefahren_vorhanden := TRUE;
			ELSE
				b_sensor_eingefahren_vorhanden := FALSE;
			END_IF
			fb_state_entry.i16_next_step := ZYL_INIT;
		END_IF

(*=======================================================*)
	ZYL_INIT:
		IF fb_state_entry.E THEN
			fb_ton_uz_fahren.IN := FALSE;
			fb_ton_uz_endlage1.IN := FALSE;
			fb_ton_uz_endlage2.IN := FALSE;
			fb_ton_uz_endlage3.IN := FALSE;
			fb_ton_uz_sensor1.IN := FALSE;
			fb_ton_uz_sensor2.IN := FALSE;
			fb_ton_uz_sensor3.IN := FALSE;
			st_tzk.fb_ton_tzk.IN	 := FALSE;
			fb_ton_einausfahren.IN := FALSE;
			fb_ton_quitt.IN := FALSE;
			a_ventil_ausfahren := FALSE;
			a_ventil_einfahren	:= FALSE;
			st_ctrl_out.b_fehler := FALSE;
			st_ctrl_out.b_eingefahren := FALSE;
			st_ctrl_out.b_ausgefahren := FALSE;
			st_ctrl_out.b_gestoppt := FALSE;
			st_ctrl_out.b_ohne_luft := FALSE;
			st_sm.b_zeit_ausfahren1:= FALSE;
			st_sm.b_zeit_einfahren1:= FALSE;
			st_sm.b_endlage1	:= FALSE;
			st_sm.b_sensor1:= FALSE;
			st_sm.b_zeit_ausfahren2 := FALSE;
			st_sm.b_zeit_einfahren2 := FALSE;
			st_sm.b_endlage2	:= FALSE;
			st_sm.b_sensor2 := FALSE;
			st_sm.b_zeit_ausfahren3 := FALSE;
			st_sm.b_zeit_einfahren3 := FALSE;
			st_sm.b_endlage3	:= FALSE;
			st_sm.b_sensor3 := FALSE;
			st_sm.b_winkel_ausfahren1:= FALSE;
			st_sm.b_winkel_einfahren1:= FALSE;
			st_sm.b_winkel_ausfahren2 := FALSE;
			st_sm.b_winkel_einfahren2 := FALSE;
			st_sm.b_winkel_ausfahren3 := FALSE;
			st_sm.b_winkel_einfahren3 := FALSE;
			st_sm.b_zyltyp_nicht_definiert := FALSE;
			st_sm.b_reserve1:= FALSE;
			b_direkttaste_ausfahren := FALSE;
			b_direkttaste_mittefahren := FALSE;
			b_direkttaste_einfahren	 := FALSE;
			b_zustand_uw_nocken_einfahren := FALSE;
			b_zustand_uw_nocken_ausfahren := FALSE;
		END_IF

		(*-----------------------Weiterschaltbedingungen----------------------------*)
		IF e_druckwaechter THEN
			CASE i16_anzahl_sensoren OF
			0:
				fb_state_entry.i16_next_step := GESTOPPT;

			1:
				IF b_nockengesteuert THEN
					IF bw_nocken_zylinder_einfahren THEN
						fb_state_entry.i16_next_step := BEWEGUNG_EINFAHREN;
					ELSIF bw_nocken_zylinder_ausfahren THEN
						fb_state_entry.i16_next_step := BEWEGUNG_AUSFAHREN;
					ELSE
						fb_state_entry.i16_next_step := GESTOPPT;
					END_IF
				ELSE
					IF  b_sensor_ausgefahren_vorhanden THEN
						IF NOT e_sensor1_ausgefahren THEN
							fb_state_entry.i16_next_step := BEWEGUNG_EINFAHREN;
						ELSIF e_sensor1_ausgefahren THEN
							fb_state_entry.i16_next_step := BEWEGUNG_AUSFAHREN;
						ELSE
							fb_state_entry.i16_next_step := GESTOPPT;
						END_IF
					ELSIF  b_sensor_eingefahren_vorhanden THEN
						IF e_sensor1_eingefahren THEN
							fb_state_entry.i16_next_step := BEWEGUNG_EINFAHREN;
						ELSIF NOT e_sensor1_eingefahren THEN
							fb_state_entry.i16_next_step := BEWEGUNG_AUSFAHREN;
						ELSE
							fb_state_entry.i16_next_step := GESTOPPT;
						END_IF
					END_IF
				END_IF

			2:
				IF b_nockengesteuert THEN
					IF bw_nocken_zylinder_einfahren THEN
						fb_state_entry.i16_next_step := BEWEGUNG_EINFAHREN;
					ELSIF bw_nocken_zylinder_ausfahren THEN
						fb_state_entry.i16_next_step := BEWEGUNG_AUSFAHREN;
					ELSE
						fb_state_entry.i16_next_step := GESTOPPT;
					END_IF
				ELSE
					IF b_sensor_eingefahren_vorhanden AND b_sensor_ausgefahren_vorhanden THEN
						IF e_sensor1_eingefahren THEN
							fb_state_entry.i16_next_step := BEWEGUNG_EINFAHREN;
						ELSIF e_sensor1_ausgefahren THEN
							fb_state_entry.i16_next_step := BEWEGUNG_AUSFAHREN;
						ELSE
							fb_state_entry.i16_next_step := GESTOPPT;
						END_IF
					ELSIF b_sensor_ausgefahren_vorhanden THEN
						IF NOT e_sensor1_ausgefahren AND NOT  e_sensor2_ausgefahren THEN
							fb_state_entry.i16_next_step := BEWEGUNG_EINFAHREN;
						ELSIF e_sensor1_ausgefahren OR e_sensor2_ausgefahren THEN
							fb_state_entry.i16_next_step := BEWEGUNG_AUSFAHREN;
						ELSE
							fb_state_entry.i16_next_step := GESTOPPT;
						END_IF
					ELSIF b_sensor_eingefahren_vorhanden THEN
						IF e_sensor1_eingefahren OR  e_sensor2_eingefahren THEN
							fb_state_entry.i16_next_step := BEWEGUNG_EINFAHREN;
						ELSIF NOT e_sensor1_eingefahren AND NOT e_sensor2_eingefahren THEN
							fb_state_entry.i16_next_step := BEWEGUNG_AUSFAHREN;
						ELSE
							fb_state_entry.i16_next_step := GESTOPPT;
						END_IF
					END_IF
				END_IF

			3:
				IF b_nockengesteuert THEN
					IF bw_nocken_zylinder_einfahren THEN
						fb_state_entry.i16_next_step := BEWEGUNG_EINFAHREN;
					ELSIF bw_nocken_zylinder_ausfahren THEN
						fb_state_entry.i16_next_step := BEWEGUNG_AUSFAHREN;
					ELSE
						fb_state_entry.i16_next_step := GESTOPPT;
					END_IF
				ELSE
					IF e_sensor1_eingefahren THEN
						fb_state_entry.i16_next_step := BEWEGUNG_EINFAHREN;
					ELSIF e_sensor1_ausgefahren THEN
						fb_state_entry.i16_next_step := BEWEGUNG_AUSFAHREN;
					ELSE
						fb_state_entry.i16_next_step := GESTOPPT;
					END_IF
				END_IF

			4:
				IF b_nockengesteuert THEN
					IF bw_nocken_zylinder_einfahren THEN
						fb_state_entry.i16_next_step := BEWEGUNG_EINFAHREN;
					ELSIF bw_nocken_zylinder_ausfahren THEN
						fb_state_entry.i16_next_step := BEWEGUNG_AUSFAHREN;
					ELSE
						fb_state_entry.i16_next_step := GESTOPPT;
					END_IF
				ELSE
					IF e_sensor1_eingefahren AND e_sensor2_eingefahren THEN
						fb_state_entry.i16_next_step := BEWEGUNG_EINFAHREN;
					ELSIF e_sensor1_ausgefahren AND e_sensor2_ausgefahren THEN
						fb_state_entry.i16_next_step := BEWEGUNG_AUSFAHREN;
					ELSE
						fb_state_entry.i16_next_step := GESTOPPT;
					END_IF
				END_IF

			6:
				IF b_nockengesteuert THEN
					IF bw_nocken_zylinder_einfahren THEN
						fb_state_entry.i16_next_step := BEWEGUNG_EINFAHREN;
					ELSIF bw_nocken_zylinder_ausfahren THEN
						fb_state_entry.i16_next_step := BEWEGUNG_AUSFAHREN;
					ELSE
						fb_state_entry.i16_next_step := GESTOPPT;
					END_IF
				ELSE
					IF e_sensor1_eingefahren AND e_sensor2_eingefahren AND e_sensor3_eingefahren THEN
						fb_state_entry.i16_next_step := BEWEGUNG_EINFAHREN;
					ELSIF e_sensor1_ausgefahren AND e_sensor2_ausgefahren AND e_sensor3_ausgefahren THEN
						fb_state_entry.i16_next_step := BEWEGUNG_AUSFAHREN;
					ELSE
						fb_state_entry.i16_next_step := GESTOPPT;
					END_IF
				END_IF
			END_CASE
		END_IF

(*=======================================================*)
	GESTOPPT:
		IF fb_state_entry.E THEN
			a_ventil_ausfahren := FALSE;
			a_ventil_einfahren	:= FALSE;
			st_ctrl_out.b_gestoppt := TRUE;
			st_ctrl_out.b_eingefahren := FALSE;
			st_ctrl_out.b_ausgefahren := FALSE;
			st_ctrl_out.b_ohne_luft := FALSE;
			st_ctrl_out.b_fehler := FALSE;
			b_zustand_uw_nocken_einfahren := FALSE;
			b_zustand_uw_nocken_ausfahren := FALSE;
		END_IF

		(*-----------------------Weiterschaltbedingungen----------------------------*)
		CASE i16_betriebsart OF
		KEINE:
			;
		AUTO, TIPPEN, DUMMY, PSEUDO:
			IF 	(st_ctrl_in.b_ausfahren AND
				NOT bw_nocken_zylinder_ausfahren AND
				NOT b_ibn_zylinder_ausfahren AND
				NOT b_direkttaste_ausfahren AND
				NOT e_taste_ausfahren) OR
				(NOT st_ctrl_in.b_ausfahren AND
				bw_nocken_zylinder_ausfahren AND
				NOT b_ibn_zylinder_ausfahren AND
				NOT b_direkttaste_ausfahren AND
				NOT e_taste_ausfahren) OR
				(NOT st_ctrl_in.b_ausfahren AND
				NOT bw_nocken_zylinder_ausfahren AND
				b_ibn_zylinder_ausfahren AND
				NOT b_direkttaste_ausfahren AND
				NOT e_taste_ausfahren)
				THEN
					fb_state_entry.i16_next_step := BEWEGUNG_AUSFAHREN;

			ELSIF	(st_ctrl_in.b_einfahren AND
					NOT bw_nocken_zylinder_einfahren AND
					NOT b_ibn_zylinder_einfahren AND
					NOT b_direkttaste_einfahren AND
					NOT e_taste_einfahren) OR
					(NOT st_ctrl_in.b_einfahren AND
					bw_nocken_zylinder_einfahren AND
					NOT b_ibn_zylinder_einfahren AND
					NOT b_direkttaste_einfahren AND
					NOT e_taste_einfahren) OR
					(NOT st_ctrl_in.b_einfahren AND
					NOT bw_nocken_zylinder_einfahren AND
					b_ibn_zylinder_einfahren AND
					NOT b_direkttaste_einfahren AND
					NOT e_taste_einfahren)
					THEN
						fb_state_entry.i16_next_step := BEWEGUNG_EINFAHREN;

			ELSIF	st_ctrl_in.b_luftlos AND
					NOT bw_nocken_zylinder_einfahren AND
					NOT b_ibn_zylinder_einfahren AND
					NOT b_direkttaste_einfahren AND
					NOT e_taste_einfahren AND
					NOT bw_nocken_zylinder_ausfahren AND
					NOT b_ibn_zylinder_ausfahren AND
					NOT b_direkttaste_ausfahren AND
					NOT e_taste_ausfahren
					THEN
						fb_state_entry.i16_next_step := LUFTLOS;
			END_IF
		HAND:
			IF	(st_visu.i16_nr_zyl_im_handbetrieb = st_config.i16_identnummer AND (st_visu.b_taste_ausfahren OR e_taste_ausfahren)) OR
				(bw_nocken_zylinder_ausfahren AND b_nockengesteuert AND b_masterachse_hand_dialog_aktiv)
				THEN
					fb_state_entry.i16_next_step := BEWEGUNG_AUSFAHREN;

			ELSIF	(st_visu.i16_nr_zyl_im_handbetrieb = st_config.i16_identnummer AND (st_visu.b_taste_einfahren OR e_taste_einfahren)) OR
					(bw_nocken_zylinder_einfahren AND b_nockengesteuert AND b_masterachse_hand_dialog_aktiv)
					THEN
						fb_state_entry.i16_next_step := BEWEGUNG_EINFAHREN;
			END_IF
		END_CASE

(*=======================================================*)
	EINGEFAHREN:
		IF fb_state_entry.E THEN
			st_ctrl_out.b_gestoppt := FALSE;
			st_ctrl_out.b_ausgefahren := FALSE;
			st_ctrl_out.b_ohne_luft := FALSE;
			fb_ton_einausfahren.IN := FALSE;
			fb_ton_uz_fahren.IN := FALSE;
			fb_ton_uz_sensor1.IN := FALSE;
			fb_ton_uz_sensor2.IN := FALSE;
			fb_ton_uz_sensor3.IN := FALSE;
			st_tzk.fb_ton_tzk.IN := FALSE;
			a_ventil_einfahren := TRUE;
			b_zustand_uw_nocken_einfahren := FALSE;
			IF NOT b_mit_tzk THEN
				st_ctrl_out.b_eingefahren := TRUE;
			END_IF
		END_IF

		IF st_ctrl_in.b_einfahren THEN	(* Messagewiederholung wenn der Zylinder sich schon im gewünschten Zustand befindet*)
			st_ctrl_out.b_eingefahren := TRUE;
		END_IF
	
		(*-----------------------Weiterschaltbedingungen----------------------------*)
		CASE i16_betriebsart OF
		KEINE:
			;
		AUTO, TIPPEN, DUMMY, PSEUDO:
			IF 	(st_ctrl_in.b_ausfahren AND
				NOT bw_nocken_zylinder_ausfahren AND
				NOT b_ibn_zylinder_ausfahren AND
				NOT b_direkttaste_ausfahren AND
				NOT e_taste_ausfahren) OR
				(NOT st_ctrl_in.b_ausfahren AND
				bw_nocken_zylinder_ausfahren  AND
				NOT b_ibn_zylinder_ausfahren AND
				NOT b_direkttaste_ausfahren AND
				NOT e_taste_ausfahren) OR
				(NOT st_ctrl_in.b_ausfahren AND
				NOT bw_nocken_zylinder_ausfahren AND
				b_ibn_zylinder_ausfahren AND
				NOT b_direkttaste_ausfahren AND
				NOT e_taste_ausfahren)
				THEN
					IF i16_anzahl_sensoren >= 1AND b_sensor_ausgefahren_vorhanden AND b_mit_tzk THEN
						st_tzk.t_ausfahrzeit_kompensiert := (st_tzk.t_ausfahrzeit * st_config.i16_tzk_faktor_ausfahren) / 100;
					END_IF
					fb_state_entry.i16_next_step := BEWEGUNG_AUSFAHREN;

			ELSIF	st_ctrl_in.b_luftlos AND
					NOT bw_nocken_zylinder_einfahren AND
					NOT b_ibn_zylinder_einfahren AND
					NOT b_direkttaste_einfahren AND
					NOT e_taste_einfahren AND
					NOT bw_nocken_zylinder_ausfahren AND
					NOT b_ibn_zylinder_ausfahren AND
					NOT b_direkttaste_ausfahren AND
					NOT e_taste_ausfahren
					THEN
						fb_state_entry.i16_next_step := LUFTLOS;
			END_IF
		HAND:
			IF	(st_visu.i16_nr_zyl_im_handbetrieb = st_config.i16_identnummer AND (st_visu.b_taste_ausfahren OR e_taste_ausfahren)) OR
				(bw_nocken_zylinder_ausfahren AND b_nockengesteuert AND b_masterachse_hand_dialog_aktiv)
				THEN
					IF i16_anzahl_sensoren >= 1AND b_sensor_ausgefahren_vorhanden AND b_mit_tzk THEN
						st_tzk.t_ausfahrzeit_kompensiert := (st_tzk.t_ausfahrzeit * st_config.i16_tzk_faktor_ausfahren) / 100;
					END_IF
					fb_state_entry.i16_next_step := BEWEGUNG_AUSFAHREN;
			END_IF
		END_CASE

		(* Überwachung auf Endlagenfehler *)
		IF i16_betriebsart <> HAND AND st_config.b_aktiv THEN
			CASE i16_anzahl_sensoren OF
				1,2,3:	(* Alle Zylinder mit mindestens einem Sensor für EINGEFAHREN *)
					IF b_sensor_eingefahren_vorhanden AND	st_config.b_endlage1_aktiv AND NOT e_sensor1_eingefahren THEN
						fb_ton_uz_endlage1.IN := TRUE;
						IF fb_ton_uz_endlage1.Q THEN
							st_sm.b_endlage1 := TRUE;
							fb_state_entry.i16_next_step := ZYL_FEHLER;
						END_IF
					ELSE
						fb_ton_uz_endlage1.IN := FALSE;
					END_IF
	
				4:	(* Alle Zylinder mit 2 Sensoren für EINGEFAHREN *)
					IF b_sensor_eingefahren_vorhanden AND st_config.b_endlage1_aktiv AND NOT e_sensor1_eingefahren THEN
						fb_ton_uz_endlage1.IN := TRUE;
						IF fb_ton_uz_endlage1.Q THEN
							st_sm.b_endlage1 := TRUE;
							fb_state_entry.i16_next_step := ZYL_FEHLER;
						END_IF
					ELSE
						fb_ton_uz_endlage1.IN := FALSE;
					END_IF
					IF b_sensor_eingefahren_vorhanden AND st_config.b_endlage2_aktiv AND NOT e_sensor2_eingefahren THEN
						fb_ton_uz_endlage2.IN := TRUE;
						IF fb_ton_uz_endlage2.Q THEN
							st_sm.b_endlage2 := TRUE;
							fb_state_entry.i16_next_step := ZYL_FEHLER;
						END_IF
					ELSE
						fb_ton_uz_endlage2.IN := FALSE;
					END_IF
	
				6:	(* Alle Zylinder mit 3 Sensoren für EINGEFAHREN *)
					IF b_sensor_eingefahren_vorhanden AND st_config.b_endlage1_aktiv AND NOT e_sensor1_eingefahren THEN
						fb_ton_uz_endlage1.IN := TRUE;
						IF fb_ton_uz_endlage1.Q THEN
							st_sm.b_endlage1 := TRUE;
							fb_state_entry.i16_next_step := ZYL_FEHLER;
						END_IF
					ELSE
						fb_ton_uz_endlage1.IN := FALSE;
					END_IF
					IF b_sensor_eingefahren_vorhanden AND st_config.b_endlage2_aktiv AND NOT e_sensor2_eingefahren THEN
						fb_ton_uz_endlage2.IN := TRUE;
						IF fb_ton_uz_endlage2.Q THEN
							st_sm.b_endlage2 := TRUE;
							fb_state_entry.i16_next_step := ZYL_FEHLER;
						END_IF
					ELSE
						fb_ton_uz_endlage2.IN := FALSE;
					END_IF
					IF b_sensor_eingefahren_vorhanden AND st_config.b_endlage3_aktiv AND NOT e_sensor3_eingefahren THEN
						fb_ton_uz_endlage3.IN := TRUE;
						IF fb_ton_uz_endlage3.Q THEN
							st_sm.b_endlage3 := TRUE;
							fb_state_entry.i16_next_step := ZYL_FEHLER;
						END_IF
					ELSE
						fb_ton_uz_endlage3.IN := FALSE;
					END_IF
			END_CASE
		END_IF

(*=======================================================*)
	BEWEGUNG_AUSFAHREN:
		IF fb_state_entry.E THEN
			st_ctrl_out.b_gestoppt := FALSE;
			st_ctrl_out.b_eingefahren := FALSE;
			st_ctrl_out.b_ausgefahren := FALSE;
			st_ctrl_out.b_ohne_luft := FALSE;
			st_ctrl_out.b_fehler := FALSE;
			a_ventil_einfahren := FALSE;
			a_ventil_ausfahren := TRUE;
			fb_ton_uz_fahren.IN := TRUE;
			fb_ton_einausfahren.IN := TRUE;
			fb_ton_uz_endlage1.IN := FALSE;
			fb_ton_uz_endlage2.IN := FALSE;
			fb_ton_uz_endlage3.IN := FALSE;
			st_sm.b_zeit_ausfahren1:= FALSE;
			st_sm.b_zeit_einfahren1:= FALSE;
			st_sm.b_endlage1	:= FALSE;
			st_sm.b_sensor1:= FALSE;
			st_sm.b_zeit_ausfahren2 := FALSE;
			st_sm.b_zeit_einfahren2 := FALSE;
			st_sm.b_endlage2	:= FALSE;
			st_sm.b_sensor2 := FALSE;
			st_sm.b_zeit_ausfahren3 := FALSE;
			st_sm.b_zeit_einfahren3 := FALSE;
			st_sm.b_endlage3	:= FALSE;
			st_sm.b_sensor3 := FALSE;
			st_sm.b_winkel_ausfahren1:= FALSE;
			st_sm.b_winkel_einfahren1:= FALSE;
			st_sm.b_winkel_ausfahren2 := FALSE;
			st_sm.b_winkel_einfahren2 := FALSE;
			st_sm.b_winkel_ausfahren3 := FALSE;
			st_sm.b_winkel_einfahren3 := FALSE;
			st_sm.b_zyltyp_nicht_definiert := FALSE;
			st_sm.b_reserve1:= FALSE;
			(* Verhindere die sofortige Fehlerauslösung, wenn Überwachungsnocken bei Stateentry schon vorhanden ist *)
			IF uw_nocken_zylinder_ausfahren THEN
				b_zustand_uw_nocken_ausfahren := TRUE;
			END_IF
		END_IF

		(* Fehlermeldung für nockengesteuerte Zylinder wieder freischalten *)
		IF fb_ton_uz_fahren.Q THEN
			b_zustand_uw_nocken_ausfahren := FALSE;
		END_IF

		CASE i16_betriebsart OF
		KEINE:
			;
		AUTO, TIPPEN, DUMMY, PSEUDO:
			IF	(st_ctrl_in.b_einfahren AND
				NOT bw_nocken_zylinder_einfahren AND
				NOT b_ibn_zylinder_einfahren AND
				NOT b_direkttaste_einfahren AND
				NOT e_taste_einfahren) OR
				(NOT st_ctrl_in.b_einfahren AND
				bw_nocken_zylinder_einfahren AND
				NOT b_ibn_zylinder_einfahren AND
				NOT b_direkttaste_einfahren AND
				NOT e_taste_einfahren) OR
				(NOT st_ctrl_in.b_einfahren AND
				NOT bw_nocken_zylinder_einfahren AND
				b_ibn_zylinder_einfahren AND
				NOT b_direkttaste_einfahren AND
				NOT e_taste_einfahren)
				THEN
					IF i16_anzahl_sensoren >= 1AND b_sensor_eingefahren_vorhanden AND b_mit_tzk THEN
						st_tzk.t_einfahrzeit_kompensiert := (st_tzk.t_einfahrzeit * st_config.i16_tzk_faktor_einfahren) / 100;
					END_IF
					fb_state_entry.i16_next_step := BEWEGUNG_EINFAHREN;
			END_IF
		HAND:
			IF	(st_visu.i16_nr_zyl_im_handbetrieb = st_config.i16_identnummer AND (st_visu.b_taste_einfahren OR e_taste_einfahren)) OR
				(bw_nocken_zylinder_einfahren AND b_nockengesteuert AND b_masterachse_hand_dialog_aktiv)
				THEN
					IF i16_anzahl_sensoren >= 1AND b_sensor_eingefahren_vorhanden AND b_mit_tzk THEN
						st_tzk.t_einfahrzeit_kompensiert := (st_tzk.t_einfahrzeit * st_config.i16_tzk_faktor_einfahren) / 100;
					END_IF
					fb_state_entry.i16_next_step := BEWEGUNG_EINFAHREN;
			END_IF
		END_CASE

		(* Totzeitkompensation mit Plausibilitätscheck der ermittelten Kompensationszeit *)
		IF	i16_anzahl_sensoren >= 1AND
			b_mit_tzk AND
			b_sensor_ausgefahren_vorhanden AND
			st_tzk.t_ausfahrzeit_kompensiert < st_tzk.t_ausfahrzeit
			THEN
				st_tzk.fb_ton_tzk.PT := st_tzk.t_ausfahrzeit_kompensiert ;
				st_tzk.fb_ton_tzk.IN := TRUE;
				(* Totzeit ist abgelaufen -> vorzeitig "ausgefahren" melden*)
				IF st_tzk.fb_ton_tzk.Q THEN
					st_ctrl_out.b_ausgefahren := TRUE;
				END_IF
		END_IF

		(*-----------------------Weiterschaltbedingungen----------------------------*)
		(* Bedingungen für Zylinder ist ausgefahren und Fehlervorkommen*)
		(* Die Sensorkonfiguration "vorhanden" ist nur für die Fälle 1, 2 von Bedeutung wegen Sonderzylinder *)
		CASE i16_anzahl_sensoren OF
			0:
				IF fb_ton_einausfahren.Q THEN
					fb_state_entry.i16_next_step := AUSGEFAHREN;
				END_IF

			1:
				IF b_sensor_ausgefahren_vorhanden THEN
					IF e_sensor1_ausgefahren THEN
						fb_state_entry.i16_next_step := AUSGEFAHREN;
					ELSE
						IF i16_betriebsart <> HAND AND st_config.b_aktiv THEN
							(* Zeitüberwachung *)
							IF fb_ton_uz_fahren.Q AND (NOT b_nockengesteuert OR b_no_gesteuert_im_norm_betrieb) THEN
								st_sm.b_zeit_ausfahren1 := TRUE;
								fb_state_entry.i16_next_step := ZYL_FEHLER;
							(* Winkelüberwachung *)
							ELSIF uw_nocken_zylinder_ausfahren AND b_nockengesteuert AND NOT b_no_gesteuert_im_norm_betrieb AND NOT b_zustand_uw_nocken_ausfahren THEN
								st_sm.b_winkel_ausfahren1 := TRUE;
								fb_state_entry.i16_next_step := ZYL_FEHLER;
							END_IF
						END_IF
					END_IF
				ELSIF b_sensor_eingefahren_vorhanden THEN
					IF  NOT e_sensor1_eingefahren THEN
						fb_state_entry.i16_next_step := AUSGEFAHREN;
					ELSE
						IF i16_betriebsart <> HAND AND st_config.b_aktiv THEN
							(* Zeitüberwachung *)
							IF fb_ton_uz_fahren.Q AND (NOT b_nockengesteuert OR b_no_gesteuert_im_norm_betrieb) THEN
								st_sm.b_zeit_ausfahren1 := TRUE;
								fb_state_entry.i16_next_step := ZYL_FEHLER;
							(* Winkelüberwachung *)
							ELSIF uw_nocken_zylinder_ausfahren AND b_nockengesteuert AND NOT b_no_gesteuert_im_norm_betrieb AND NOT b_zustand_uw_nocken_ausfahren THEN
								st_sm.b_winkel_ausfahren1 := TRUE;
								fb_state_entry.i16_next_step := ZYL_FEHLER;
							END_IF
						END_IF
					END_IF
				END_IF

			2:
				IF b_sensor_eingefahren_vorhanden AND b_sensor_ausgefahren_vorhanden THEN
					IF e_sensor1_ausgefahren AND NOT e_sensor1_eingefahren THEN
						fb_state_entry.i16_next_step := AUSGEFAHREN;
					ELSE
						IF i16_betriebsart <> HAND AND st_config.b_aktiv THEN
							(* Zeitüberwachung *)
							IF fb_ton_uz_fahren.Q AND (NOT b_nockengesteuert OR b_no_gesteuert_im_norm_betrieb) THEN
								st_sm.b_zeit_ausfahren1 := TRUE;
								fb_state_entry.i16_next_step := ZYL_FEHLER;
							(* Winkelüberwachung *)
							ELSIF uw_nocken_zylinder_ausfahren AND b_nockengesteuert AND NOT b_no_gesteuert_im_norm_betrieb AND NOT b_zustand_uw_nocken_ausfahren THEN
								st_sm.b_winkel_ausfahren1 := TRUE;
								fb_state_entry.i16_next_step := ZYL_FEHLER;
							END_IF
						END_IF
					END_IF
				ELSIF b_sensor_eingefahren_vorhanden THEN
					IF NOT e_sensor1_eingefahren AND NOT e_sensor2_eingefahren THEN
						fb_state_entry.i16_next_step := AUSGEFAHREN;
					ELSE
						IF i16_betriebsart <> HAND AND st_config.b_aktiv THEN
							(* Zeitüberwachung *)
							IF fb_ton_uz_fahren.Q AND (NOT b_nockengesteuert OR b_no_gesteuert_im_norm_betrieb) THEN
								IF e_sensor1_eingefahren THEN
									st_sm.b_zeit_ausfahren1 := TRUE;
								END_IF
								IF e_sensor2_eingefahren THEN
									st_sm.b_zeit_ausfahren2 := TRUE;
								END_IF
								fb_state_entry.i16_next_step := ZYL_FEHLER;
							(* Winkelüberwachung *)
							ELSIF uw_nocken_zylinder_ausfahren AND b_nockengesteuert AND NOT b_no_gesteuert_im_norm_betrieb AND NOT b_zustand_uw_nocken_ausfahren THEN
								IF e_sensor1_eingefahren THEN
									st_sm.b_winkel_ausfahren1 := TRUE;
								END_IF
								IF e_sensor2_eingefahren THEN
									st_sm.b_winkel_ausfahren2 := TRUE;
								END_IF
								fb_state_entry.i16_next_step := ZYL_FEHLER;
							END_IF
						END_IF
					END_IF
				ELSIF  b_sensor_ausgefahren_vorhanden THEN
					IF e_sensor1_ausgefahren AND e_sensor2_ausgefahren THEN
						fb_state_entry.i16_next_step := AUSGEFAHREN;
					ELSE
						IF i16_betriebsart <> HAND AND st_config.b_aktiv THEN
							(* Zeitüberwachung *)
							IF fb_ton_uz_fahren.Q AND (NOT b_nockengesteuert OR b_no_gesteuert_im_norm_betrieb) THEN
								IF NOT e_sensor1_ausgefahren THEN
									st_sm.b_zeit_ausfahren1 := TRUE;
								END_IF
								IF NOT e_sensor2_ausgefahren THEN
									st_sm.b_zeit_ausfahren2 := TRUE;
								END_IF
								fb_state_entry.i16_next_step := ZYL_FEHLER;
							(* Winkelüberwachung *)
							ELSIF uw_nocken_zylinder_ausfahren AND b_nockengesteuert AND NOT b_no_gesteuert_im_norm_betrieb AND NOT b_zustand_uw_nocken_ausfahren THEN
								IF NOT e_sensor1_ausgefahren THEN
									st_sm.b_winkel_ausfahren1 := TRUE;
								END_IF
								IF NOT e_sensor2_ausgefahren THEN
									st_sm.b_winkel_ausfahren2 := TRUE;
								END_IF
								fb_state_entry.i16_next_step := ZYL_FEHLER;
							END_IF
						END_IF
					END_IF
				END_IF
				IF i16_betriebsart <> HAND AND st_config.b_aktiv THEN
					(* Überwachung auf Sensorfehler *)
					IF e_sensor1_ausgefahren  AND e_sensor1_eingefahren  AND st_config.b_sensor1_aktiv THEN
						fb_ton_uz_sensor1.IN := TRUE;
						IF fb_ton_uz_sensor1.Q THEN
							st_sm.b_sensor1 := TRUE;
							fb_state_entry.i16_next_step := ZYL_FEHLER;
						END_IF
					ELSE
						fb_ton_uz_sensor1.IN := FALSE;
					END_IF
				END_IF

